// TwinCAT 3 PLC project PLC
// ProgramVersion: 3.1.4023.0
// libraries:
//   SPT Base Types, * (Beckhoff Automation LLC)
//   SPT XTS, * (Beckhoff Automation LLC)
//   Tc2_Standard, * (Beckhoff Automation GmbH)
//   Tc2_System, * (Beckhoff Automation GmbH)
//   Tc3_Module, * (Beckhoff Automation GmbH)
//   Tc3_PackML_V2, * (Beckhoff Automation GmbH)
//   Tc3_XTS_Utility, * (Beckhoff Automation GmbH)
// project tree:
//   / FB_Machine.TcPOU, PlcTask.TcTTO
//   POUs/ MAIN.TcPOU
// real-time tasks:
//   TASK XTS Task 1: cycle T#250us, priority 1, ADS port 350
//   TASK Job Task: cycle default, priority 32
//   TASK PlcTask: cycle T#10ms, priority 20, ADS port 351
// motion (NC):
//   TASK NC-Task 1: cycle T#2ms, priority 4, ADS port 501
//   TASK NC-Task 1 SVB: cycle T#10ms, priority 8, ADS port 511
//   AXIS Mover Axis 1 (id 1)
//     Dynamic: AccelerationMaximum=80000, DecelerationMaximum=80000, Acceleration=20000, Deceleration=20000, Jerk=200000
//     Velo: Maximum=4000
//     PositionAreaControl: Enable=false
//     TargetPosControl: Enable=false
//     OtherSettings: AllowMotionCmdToSlave=true, AllowMotionCmdToExtSetGenAxis=true
//     encoder EncType=28
//       EncPara: ModuloFactor=3000, ToleranceWndModuloStart=0.2, MaxCount=#xffffffff
//     drive DrvType=22
//       DrvPara: MaxCount=#xffffffff, DriveControlDWord=#x00000100
//         Analog: VeloReferenz=4200, TorqueSetpointScale=10
//         TimeComp: TaskDelayCycles=1
//     controller CtrType=1
//       CtrPara: PriorControlFactor=1
//         PosDiffControl: Range=10
//         Observer: BandWidth=20
//   AXIS Mover Axis 2 (id 2)
//     Dynamic: AccelerationMaximum=80000, DecelerationMaximum=80000, Acceleration=20000, Deceleration=20000, Jerk=200000
//     Velo: Maximum=4000
//     PositionAreaControl: Enable=false
//     TargetPosControl: Enable=false
//     OtherSettings: AllowMotionCmdToSlave=true, AllowMotionCmdToExtSetGenAxis=true
//     encoder EncType=28
//       EncPara: ModuloFactor=3000, ToleranceWndModuloStart=0.2, MaxCount=#xffffffff
//     drive DrvType=22
//       DrvPara: MaxCount=#xffffffff, DriveControlDWord=#x00000100
//         Analog: VeloReferenz=4200, TorqueSetpointScale=10
//         TimeComp: TaskDelayCycles=1
//     controller CtrType=1
//       CtrPara: PriorControlFactor=1
//         PosDiffControl: Range=10
//         Observer: BandWidth=20
//   AXIS Mover Axis 3 (id 3)
//     Dynamic: AccelerationMaximum=80000, DecelerationMaximum=80000, Acceleration=20000, Deceleration=20000, Jerk=200000
//     Velo: Maximum=4000
//     PositionAreaControl: Enable=false
//     TargetPosControl: Enable=false
//     OtherSettings: AllowMotionCmdToSlave=true, AllowMotionCmdToExtSetGenAxis=true
//     encoder EncType=28
//       EncPara: ModuloFactor=3000, ToleranceWndModuloStart=0.2, MaxCount=#xffffffff
//     drive DrvType=22
//       DrvPara: MaxCount=#xffffffff, DriveControlDWord=#x00000100
//         Analog: VeloReferenz=4200, TorqueSetpointScale=10
//         TimeComp: TaskDelayCycles=1
//     controller CtrType=1
//       CtrPara: PriorControlFactor=1
//         PosDiffControl: Range=10
//         Observer: BandWidth=20
//   AXIS Mover Axis 4 (id 4)
//     Dynamic: AccelerationMaximum=80000, DecelerationMaximum=80000, Acceleration=20000, Deceleration=20000, Jerk=200000
//     Velo: Maximum=4000
//     PositionAreaControl: Enable=false
//     TargetPosControl: Enable=false
//     OtherSettings: AllowMotionCmdToSlave=true, AllowMotionCmdToExtSetGenAxis=true
//     encoder EncType=28
//       EncPara: ModuloFactor=3000, ToleranceWndModuloStart=0.2, MaxCount=#xffffffff
//     drive DrvType=22
//       DrvPara: MaxCount=#xffffffff, DriveControlDWord=#x00000100
//         Analog: VeloReferenz=4200, TorqueSetpointScale=10
//         TimeComp: TaskDelayCycles=1
//     controller CtrType=1
//       CtrPara: PriorControlFactor=1
//         PosDiffControl: Range=10
//         Observer: BandWidth=20
//   AXIS Mover Axis 5 (id 5)
//     Dynamic: AccelerationMaximum=80000, DecelerationMaximum=80000, Acceleration=20000, Deceleration=20000, Jerk=200000
//     Velo: Maximum=4000
//     PositionAreaControl: Enable=false
//     TargetPosControl: Enable=false
//     OtherSettings: AllowMotionCmdToSlave=true, AllowMotionCmdToExtSetGenAxis=true
//     encoder EncType=28
//       EncPara: ModuloFactor=3000, ToleranceWndModuloStart=0.2, MaxCount=#xffffffff
//     drive DrvType=22
//       DrvPara: MaxCount=#xffffffff, DriveControlDWord=#x00000100
//         Analog: VeloReferenz=4200, TorqueSetpointScale=10
//         TimeComp: TaskDelayCycles=1
//     controller CtrType=1
//       CtrPara: PriorControlFactor=1
//         PosDiffControl: Range=10
//         Observer: BandWidth=20
//   AXIS Mover Axis 6 (id 6)
//     Dynamic: AccelerationMaximum=80000, DecelerationMaximum=80000, Acceleration=20000, Deceleration=20000, Jerk=200000
//     Velo: Maximum=4000
//     PositionAreaControl: Enable=false
//     TargetPosControl: Enable=false
//     OtherSettings: AllowMotionCmdToSlave=true, AllowMotionCmdToExtSetGenAxis=true
//     encoder EncType=28
//       EncPara: ModuloFactor=3000, ToleranceWndModuloStart=0.2, MaxCount=#xffffffff
//     drive DrvType=22
//       DrvPara: MaxCount=#xffffffff, DriveControlDWord=#x00000100
//         Analog: VeloReferenz=4200, TorqueSetpointScale=10
//         TimeComp: TaskDelayCycles=1
//     controller CtrType=1
//       CtrPara: PriorControlFactor=1
//         PosDiffControl: Range=10
//         Observer: BandWidth=20
//   AXIS Mover Axis 7 (id 7)
//     Dynamic: AccelerationMaximum=80000, DecelerationMaximum=80000, Acceleration=20000, Deceleration=20000, Jerk=200000
//     Velo: Maximum=4000
//     PositionAreaControl: Enable=false
//     TargetPosControl: Enable=false
//     OtherSettings: AllowMotionCmdToSlave=true, AllowMotionCmdToExtSetGenAxis=true
//     encoder EncType=28
//       EncPara: ModuloFactor=3000, ToleranceWndModuloStart=0.2, MaxCount=#xffffffff
//     drive DrvType=22
//       DrvPara: MaxCount=#xffffffff, DriveControlDWord=#x00000100
//         Analog: VeloReferenz=4200, TorqueSetpointScale=10
//         TimeComp: TaskDelayCycles=1
//     controller CtrType=1
//       CtrPara: PriorControlFactor=1
//         PosDiffControl: Range=10
//         Observer: BandWidth=20
//   AXIS Mover Axis 8 (id 8)
//     Dynamic: AccelerationMaximum=80000, DecelerationMaximum=80000, Acceleration=20000, Deceleration=20000, Jerk=200000
//     Velo: Maximum=4000
//     PositionAreaControl: Enable=false
//     TargetPosControl: Enable=false
//     OtherSettings: AllowMotionCmdToSlave=true, AllowMotionCmdToExtSetGenAxis=true
//     encoder EncType=28
//       EncPara: ModuloFactor=3000, ToleranceWndModuloStart=0.2, MaxCount=#xffffffff
//     drive DrvType=22
//       DrvPara: MaxCount=#xffffffff, DriveControlDWord=#x00000100
//         Analog: VeloReferenz=4200, TorqueSetpointScale=10
//         TimeComp: TaskDelayCycles=1
//     controller CtrType=1
//       CtrPara: PriorControlFactor=1
//         PosDiffControl: Range=10
//         Observer: BandWidth=20
//   AXIS Mover Axis 9 (id 9)
//     Dynamic: AccelerationMaximum=80000, DecelerationMaximum=80000, Acceleration=20000, Deceleration=20000, Jerk=200000
//     Velo: Maximum=4000
//     PositionAreaControl: Enable=false
//     TargetPosControl: Enable=false
//     OtherSettings: AllowMotionCmdToSlave=true, AllowMotionCmdToExtSetGenAxis=true
//     encoder EncType=28
//       EncPara: ModuloFactor=3000, ToleranceWndModuloStart=0.2, MaxCount=#xffffffff
//     drive DrvType=22
//       DrvPara: MaxCount=#xffffffff, DriveControlDWord=#x00000100
//         Analog: VeloReferenz=4200, TorqueSetpointScale=10
//         TimeComp: TaskDelayCycles=1
//     controller CtrType=1
//       CtrPara: PriorControlFactor=1
//         PosDiffControl: Range=10
//         Observer: BandWidth=20
//   AXIS Mover Axis 10 (id 10)
//     Dynamic: AccelerationMaximum=80000, DecelerationMaximum=80000, Acceleration=20000, Deceleration=20000, Jerk=200000
//     Velo: Maximum=4000
//     PositionAreaControl: Enable=false
//     TargetPosControl: Enable=false
//     OtherSettings: AllowMotionCmdToSlave=true, AllowMotionCmdToExtSetGenAxis=true
//     encoder EncType=28
//       EncPara: ModuloFactor=3000, ToleranceWndModuloStart=0.2, MaxCount=#xffffffff
//     drive DrvType=22
//       DrvPara: MaxCount=#xffffffff, DriveControlDWord=#x00000100
//         Analog: VeloReferenz=4200, TorqueSetpointScale=10
//         TimeComp: TaskDelayCycles=1
//     controller CtrType=1
//       CtrPara: PriorControlFactor=1
//         PosDiffControl: Range=10
//         Observer: BandWidth=20
// I/O:
//   DEVICE Device 1 (disabled), AmsNetId 192.168.111.1.2.1
//     Term 1 (AT2001-0250) [AT2001-0250 Motor module with feed 250 mm, 48V]
//       Term 2 (AT2001-5250) [AT2001-5250 Sensor line with feed]
//     Term 3 (AT2000-0250) [AT2000-0250 Motor module 250 mm, 48V]
//       Term 4 (AT2000-5250) [AT2000-5250 Sensor line]
//     Term 5 (AT2000-0250) [AT2000-0250 Motor module 250 mm, 48V]
//       Term 6 (AT2000-5250) [AT2000-5250 Sensor line]
//     Term 7 (AT2000-0250) [AT2000-0250 Motor module 250 mm, 48V]
//       Term 8 (AT2000-5250) [AT2000-5250 Sensor line]
//     Term 9 (AT2050-0500) [AT2050-0500 Motor module, 90° clothoid, EtherCAT In, 48V]
//       Term 10 (AT2050-5500) [AT2050-5500 Sensor line 90° clothoid, EtherCAT In]
//     Term 11 (AT2050-0501) [AT2050-0501 Motor module, 90° clothoid, EtherCAT Out, 48V]
//       Term 12 (AT2050-5501) [AT2050-5501 Sensor line 90° clothoid, EtherCAT Out]
//   DEVICE Device 2 (disabled), AmsNetId 192.168.111.1.3.1
//     Term 13 (AT2001-0250) [AT2001-0250 Motor module with feed 250 mm, 48V]
//       Term 14 (AT2001-5250) [AT2001-5250 Sensor line with feed]
//     Term 15 (AT2000-0250) [AT2000-0250 Motor module 250 mm, 48V]
//       Term 16 (AT2000-5250) [AT2000-5250 Sensor line]
//     Term 17 (AT2000-0250) [AT2000-0250 Motor module 250 mm, 48V]
//       Term 18 (AT2000-5250) [AT2000-5250 Sensor line]
//     Term 19 (AT2000-0250) [AT2000-0250 Motor module 250 mm, 48V]
//       Term 20 (AT2000-5250) [AT2000-5250 Sensor line]
//     Term 21 (AT2050-0500) [AT2050-0500 Motor module, 90° clothoid, EtherCAT In, 48V]
//       Term 22 (AT2050-5500) [AT2050-5500 Sensor line 90° clothoid, EtherCAT In]
//     Term 23 (AT2050-0501) [AT2050-0501 Motor module, 90° clothoid, EtherCAT Out, 48V]
//       Term 24 (AT2050-5501) [AT2050-5501 Sensor line 90° clothoid, EtherCAT Out]
// variable links:
//   Device 1 <-> TcCOM Objects/XtsProcessingUnit 1/Part 1/Module 1
//     Term 1 (AT2001-0250)/CC Inputs/Current actual value Ch.1 <-> Data Pointer/CurrentActualValues[0]
//     Term 1 (AT2001-0250)/CC Inputs/Current actual value Ch.10 <-> Data Pointer/CurrentActualValues[9]
//     Term 1 (AT2001-0250)/CC Inputs/Current actual value Ch.11 <-> Data Pointer/CurrentActualValues[10]
//     Term 1 (AT2001-0250)/CC Inputs/Current actual value Ch.12 <-> Data Pointer/CurrentActualValues[11]
//     Term 1 (AT2001-0250)/CC Inputs/Current actual value Ch.13 <-> Data Pointer/CurrentActualValues[12]
//     Term 1 (AT2001-0250)/CC Inputs/Current actual value Ch.14 <-> Data Pointer/CurrentActualValues[13]
//     Term 1 (AT2001-0250)/CC Inputs/Current actual value Ch.15 <-> Data Pointer/CurrentActualValues[14]
//     Term 1 (AT2001-0250)/CC Inputs/Current actual value Ch.2 <-> Data Pointer/CurrentActualValues[1]
//     Term 1 (AT2001-0250)/CC Inputs/Current actual value Ch.3 <-> Data Pointer/CurrentActualValues[2]
//     Term 1 (AT2001-0250)/CC Inputs/Current actual value Ch.4 <-> Data Pointer/CurrentActualValues[3]
//     Term 1 (AT2001-0250)/CC Inputs/Current actual value Ch.5 <-> Data Pointer/CurrentActualValues[4]
//     Term 1 (AT2001-0250)/CC Inputs/Current actual value Ch.6 <-> Data Pointer/CurrentActualValues[5]
//     Term 1 (AT2001-0250)/CC Inputs/Current actual value Ch.7 <-> Data Pointer/CurrentActualValues[6]
//     Term 1 (AT2001-0250)/CC Inputs/Current actual value Ch.8 <-> Data Pointer/CurrentActualValues[7]
//     Term 1 (AT2001-0250)/CC Inputs/Current actual value Ch.9 <-> Data Pointer/CurrentActualValues[8]
//     Term 1 (AT2001-0250)/CC Inputs/Status <-> Data Pointer/Status
//     Term 1 (AT2001-0250)/CC Outputs/Control <-> Data Pointer/Control
//     Term 1 (AT2001-0250)/CC Outputs/Current setpoint value Ch.1 <-> Data Pointer/CurrentSetpointValues[0]
//     Term 1 (AT2001-0250)/CC Outputs/Current setpoint value Ch.10 <-> Data Pointer/CurrentSetpointValues[9]
//     Term 1 (AT2001-0250)/CC Outputs/Current setpoint value Ch.11 <-> Data Pointer/CurrentSetpointValues[10]
//     Term 1 (AT2001-0250)/CC Outputs/Current setpoint value Ch.12 <-> Data Pointer/CurrentSetpointValues[11]
//     Term 1 (AT2001-0250)/CC Outputs/Current setpoint value Ch.13 <-> Data Pointer/CurrentSetpointValues[12]
//     Term 1 (AT2001-0250)/CC Outputs/Current setpoint value Ch.14 <-> Data Pointer/CurrentSetpointValues[13]
//     Term 1 (AT2001-0250)/CC Outputs/Current setpoint value Ch.15 <-> Data Pointer/CurrentSetpointValues[14]
//     Term 1 (AT2001-0250)/CC Outputs/Current setpoint value Ch.2 <-> Data Pointer/CurrentSetpointValues[1]
//     Term 1 (AT2001-0250)/CC Outputs/Current setpoint value Ch.3 <-> Data Pointer/CurrentSetpointValues[2]
//     Term 1 (AT2001-0250)/CC Outputs/Current setpoint value Ch.4 <-> Data Pointer/CurrentSetpointValues[3]
//     Term 1 (AT2001-0250)/CC Outputs/Current setpoint value Ch.5 <-> Data Pointer/CurrentSetpointValues[4]
//     Term 1 (AT2001-0250)/CC Outputs/Current setpoint value Ch.6 <-> Data Pointer/CurrentSetpointValues[5]
//     Term 1 (AT2001-0250)/CC Outputs/Current setpoint value Ch.7 <-> Data Pointer/CurrentSetpointValues[6]
//     Term 1 (AT2001-0250)/CC Outputs/Current setpoint value Ch.8 <-> Data Pointer/CurrentSetpointValues[7]
//     Term 1 (AT2001-0250)/CC Outputs/Current setpoint value Ch.9 <-> Data Pointer/CurrentSetpointValues[8]
//     Term 1 (AT2001-0250)/Term 2 (AT2001-5250)/FB Inputs/Value Channel 01 <-> Data Pointer/RawPositionValues[0]
//     Term 1 (AT2001-0250)/Term 2 (AT2001-5250)/FB Inputs/Value Channel 02 <-> Data Pointer/RawPositionValues[1]
//     Term 1 (AT2001-0250)/Term 2 (AT2001-5250)/FB Inputs/Value Channel 03 <-> Data Pointer/RawPositionValues[2]
//     Term 1 (AT2001-0250)/Term 2 (AT2001-5250)/FB Inputs/Value Channel 04 <-> Data Pointer/RawPositionValues[3]
//     Term 1 (AT2001-0250)/Term 2 (AT2001-5250)/FB Inputs/Value Channel 05 <-> Data Pointer/RawPositionValues[4]
//     Term 1 (AT2001-0250)/Term 2 (AT2001-5250)/FB Inputs/Value Channel 06 <-> Data Pointer/RawPositionValues[5]
//     Term 1 (AT2001-0250)/Term 2 (AT2001-5250)/FB Inputs/Value Channel 07 <-> Data Pointer/RawPositionValues[6]
//     Term 1 (AT2001-0250)/Term 2 (AT2001-5250)/FB Inputs/Value Channel 08 <-> Data Pointer/RawPositionValues[7]
//     Term 1 (AT2001-0250)/Term 2 (AT2001-5250)/FB Inputs/Value Channel 09 <-> Data Pointer/RawPositionValues[8]
//     Term 1 (AT2001-0250)/Term 2 (AT2001-5250)/FB Inputs/Value Channel 10 <-> Data Pointer/RawPositionValues[9]
//     Term 1 (AT2001-0250)/Term 2 (AT2001-5250)/FB Inputs/Value Channel 11 <-> Data Pointer/RawPositionValues[10]
//     Term 1 (AT2001-0250)/Term 2 (AT2001-5250)/FB Inputs/Value Channel 12 <-> Data Pointer/RawPositionValues[11]
//     Term 1 (AT2001-0250)/Term 2 (AT2001-5250)/FB Inputs/Value Channel 13 <-> Data Pointer/RawPositionValues[12]
//     Term 1 (AT2001-0250)/Term 2 (AT2001-5250)/FB Inputs/Value Channel 14 <-> Data Pointer/RawPositionValues[13]
//     Term 1 (AT2001-0250)/Term 2 (AT2001-5250)/FB Inputs/Value Channel 15 <-> Data Pointer/RawPositionValues[14]
//     Term 1 (AT2001-0250)/Term 2 (AT2001-5250)/FB Inputs/Value Channel 16 <-> Data Pointer/RawPositionValues[15]
//     Term 1 (AT2001-0250)/Term 2 (AT2001-5250)/FB Inputs/Value Channel 17 <-> Data Pointer/RawPositionValues[16]
//     Term 1 (AT2001-0250)/Term 2 (AT2001-5250)/FB Inputs/Value Channel 18 <-> Data Pointer/RawPositionValues[17]
//     Term 1 (AT2001-0250)/Term 2 (AT2001-5250)/FB Inputs/Value Channel 19 <-> Data Pointer/RawPositionValues[18]
//     Term 1 (AT2001-0250)/Term 2 (AT2001-5250)/FB Inputs/Value Channel 20 <-> Data Pointer/RawPositionValues[19]
//     Term 1 (AT2001-0250)/Term 2 (AT2001-5250)/FB Inputs/Value Channel 21 <-> Data Pointer/RawPositionValues[20]
//     Term 1 (AT2001-0250)/Term 2 (AT2001-5250)/FB Inputs/Value Channel 22 <-> Data Pointer/RawPositionValues[21]
//     Term 1 (AT2001-0250)/Term 2 (AT2001-5250)/FB Inputs/Value Channel 23 <-> Data Pointer/RawPositionValues[22]
//     Term 1 (AT2001-0250)/Term 2 (AT2001-5250)/FB Inputs/Value Channel 24 <-> Data Pointer/RawPositionValues[23]
//     Term 1 (AT2001-0250)/Term 2 (AT2001-5250)/FB Inputs/Value Channel 25 <-> Data Pointer/RawPositionValues[24]
//     Term 1 (AT2001-0250)/Term 2 (AT2001-5250)/FB Inputs/Value Channel 26 <-> Data Pointer/RawPositionValues[25]
//     Term 1 (AT2001-0250)/Term 2 (AT2001-5250)/FB Inputs/Value Channel 27 <-> Data Pointer/RawPositionValues[26]
//     Term 1 (AT2001-0250)/Term 2 (AT2001-5250)/FB Inputs/Value Channel 28 <-> Data Pointer/RawPositionValues[27]
//     Term 1 (AT2001-0250)/Term 2 (AT2001-5250)/FB Inputs/Value Channel 29 <-> Data Pointer/RawPositionValues[28]
//     Term 1 (AT2001-0250)/Term 2 (AT2001-5250)/FB Inputs/Value Channel 30 <-> Data Pointer/RawPositionValues[29]
//     Term 1 (AT2001-0250)/Term 2 (AT2001-5250)/FB Inputs/Value Channel 31 <-> Data Pointer/RawPositionValues[30]
//     Term 1 (AT2001-0250)/Term 2 (AT2001-5250)/FB Inputs/Value Channel 32 <-> Data Pointer/RawPositionValues[31]
//   Device 1 <-> TcCOM Objects/XtsProcessingUnit 1/Part 1/Module 2
//     Term 3 (AT2000-0250)/CC Inputs/Current actual value Ch.1 <-> Data Pointer/CurrentActualValues[0]
//     Term 3 (AT2000-0250)/CC Inputs/Current actual value Ch.10 <-> Data Pointer/CurrentActualValues[9]
//     Term 3 (AT2000-0250)/CC Inputs/Current actual value Ch.11 <-> Data Pointer/CurrentActualValues[10]
//     Term 3 (AT2000-0250)/CC Inputs/Current actual value Ch.12 <-> Data Pointer/CurrentActualValues[11]
//     Term 3 (AT2000-0250)/CC Inputs/Current actual value Ch.13 <-> Data Pointer/CurrentActualValues[12]
//     Term 3 (AT2000-0250)/CC Inputs/Current actual value Ch.14 <-> Data Pointer/CurrentActualValues[13]
//     Term 3 (AT2000-0250)/CC Inputs/Current actual value Ch.15 <-> Data Pointer/CurrentActualValues[14]
//     Term 3 (AT2000-0250)/CC Inputs/Current actual value Ch.2 <-> Data Pointer/CurrentActualValues[1]
//     Term 3 (AT2000-0250)/CC Inputs/Current actual value Ch.3 <-> Data Pointer/CurrentActualValues[2]
//     Term 3 (AT2000-0250)/CC Inputs/Current actual value Ch.4 <-> Data Pointer/CurrentActualValues[3]
//     Term 3 (AT2000-0250)/CC Inputs/Current actual value Ch.5 <-> Data Pointer/CurrentActualValues[4]
//     Term 3 (AT2000-0250)/CC Inputs/Current actual value Ch.6 <-> Data Pointer/CurrentActualValues[5]
//     Term 3 (AT2000-0250)/CC Inputs/Current actual value Ch.7 <-> Data Pointer/CurrentActualValues[6]
//     Term 3 (AT2000-0250)/CC Inputs/Current actual value Ch.8 <-> Data Pointer/CurrentActualValues[7]
//     Term 3 (AT2000-0250)/CC Inputs/Current actual value Ch.9 <-> Data Pointer/CurrentActualValues[8]
//     Term 3 (AT2000-0250)/CC Inputs/Status <-> Data Pointer/Status
//     Term 3 (AT2000-0250)/CC Outputs/Control <-> Data Pointer/Control
//     Term 3 (AT2000-0250)/CC Outputs/Current setpoint value Ch.1 <-> Data Pointer/CurrentSetpointValues[0]
//     Term 3 (AT2000-0250)/CC Outputs/Current setpoint value Ch.10 <-> Data Pointer/CurrentSetpointValues[9]
//     Term 3 (AT2000-0250)/CC Outputs/Current setpoint value Ch.11 <-> Data Pointer/CurrentSetpointValues[10]
//     Term 3 (AT2000-0250)/CC Outputs/Current setpoint value Ch.12 <-> Data Pointer/CurrentSetpointValues[11]
//     Term 3 (AT2000-0250)/CC Outputs/Current setpoint value Ch.13 <-> Data Pointer/CurrentSetpointValues[12]
//     Term 3 (AT2000-0250)/CC Outputs/Current setpoint value Ch.14 <-> Data Pointer/CurrentSetpointValues[13]
//     Term 3 (AT2000-0250)/CC Outputs/Current setpoint value Ch.15 <-> Data Pointer/CurrentSetpointValues[14]
//     Term 3 (AT2000-0250)/CC Outputs/Current setpoint value Ch.2 <-> Data Pointer/CurrentSetpointValues[1]
//     Term 3 (AT2000-0250)/CC Outputs/Current setpoint value Ch.3 <-> Data Pointer/CurrentSetpointValues[2]
//     Term 3 (AT2000-0250)/CC Outputs/Current setpoint value Ch.4 <-> Data Pointer/CurrentSetpointValues[3]
//     Term 3 (AT2000-0250)/CC Outputs/Current setpoint value Ch.5 <-> Data Pointer/CurrentSetpointValues[4]
//     Term 3 (AT2000-0250)/CC Outputs/Current setpoint value Ch.6 <-> Data Pointer/CurrentSetpointValues[5]
//     Term 3 (AT2000-0250)/CC Outputs/Current setpoint value Ch.7 <-> Data Pointer/CurrentSetpointValues[6]
//     Term 3 (AT2000-0250)/CC Outputs/Current setpoint value Ch.8 <-> Data Pointer/CurrentSetpointValues[7]
//     Term 3 (AT2000-0250)/CC Outputs/Current setpoint value Ch.9 <-> Data Pointer/CurrentSetpointValues[8]
//     Term 3 (AT2000-0250)/Term 4 (AT2000-5250)/FB Inputs/Value Channel 01 <-> Data Pointer/RawPositionValues[0]
//     Term 3 (AT2000-0250)/Term 4 (AT2000-5250)/FB Inputs/Value Channel 02 <-> Data Pointer/RawPositionValues[1]
//     Term 3 (AT2000-0250)/Term 4 (AT2000-5250)/FB Inputs/Value Channel 03 <-> Data Pointer/RawPositionValues[2]
//     Term 3 (AT2000-0250)/Term 4 (AT2000-5250)/FB Inputs/Value Channel 04 <-> Data Pointer/RawPositionValues[3]
//     Term 3 (AT2000-0250)/Term 4 (AT2000-5250)/FB Inputs/Value Channel 05 <-> Data Pointer/RawPositionValues[4]
//     Term 3 (AT2000-0250)/Term 4 (AT2000-5250)/FB Inputs/Value Channel 06 <-> Data Pointer/RawPositionValues[5]
//     Term 3 (AT2000-0250)/Term 4 (AT2000-5250)/FB Inputs/Value Channel 07 <-> Data Pointer/RawPositionValues[6]
//     Term 3 (AT2000-0250)/Term 4 (AT2000-5250)/FB Inputs/Value Channel 08 <-> Data Pointer/RawPositionValues[7]
//     Term 3 (AT2000-0250)/Term 4 (AT2000-5250)/FB Inputs/Value Channel 09 <-> Data Pointer/RawPositionValues[8]
//     Term 3 (AT2000-0250)/Term 4 (AT2000-5250)/FB Inputs/Value Channel 10 <-> Data Pointer/RawPositionValues[9]
//     Term 3 (AT2000-0250)/Term 4 (AT2000-5250)/FB Inputs/Value Channel 11 <-> Data Pointer/RawPositionValues[10]
//     Term 3 (AT2000-0250)/Term 4 (AT2000-5250)/FB Inputs/Value Channel 12 <-> Data Pointer/RawPositionValues[11]
//     Term 3 (AT2000-0250)/Term 4 (AT2000-5250)/FB Inputs/Value Channel 13 <-> Data Pointer/RawPositionValues[12]
//     Term 3 (AT2000-0250)/Term 4 (AT2000-5250)/FB Inputs/Value Channel 14 <-> Data Pointer/RawPositionValues[13]
//     Term 3 (AT2000-0250)/Term 4 (AT2000-5250)/FB Inputs/Value Channel 15 <-> Data Pointer/RawPositionValues[14]
//     Term 3 (AT2000-0250)/Term 4 (AT2000-5250)/FB Inputs/Value Channel 16 <-> Data Pointer/RawPositionValues[15]
//     Term 3 (AT2000-0250)/Term 4 (AT2000-5250)/FB Inputs/Value Channel 17 <-> Data Pointer/RawPositionValues[16]
//     Term 3 (AT2000-0250)/Term 4 (AT2000-5250)/FB Inputs/Value Channel 18 <-> Data Pointer/RawPositionValues[17]
//     Term 3 (AT2000-0250)/Term 4 (AT2000-5250)/FB Inputs/Value Channel 19 <-> Data Pointer/RawPositionValues[18]
//     Term 3 (AT2000-0250)/Term 4 (AT2000-5250)/FB Inputs/Value Channel 20 <-> Data Pointer/RawPositionValues[19]
//     Term 3 (AT2000-0250)/Term 4 (AT2000-5250)/FB Inputs/Value Channel 21 <-> Data Pointer/RawPositionValues[20]
//     Term 3 (AT2000-0250)/Term 4 (AT2000-5250)/FB Inputs/Value Channel 22 <-> Data Pointer/RawPositionValues[21]
//     Term 3 (AT2000-0250)/Term 4 (AT2000-5250)/FB Inputs/Value Channel 23 <-> Data Pointer/RawPositionValues[22]
//     Term 3 (AT2000-0250)/Term 4 (AT2000-5250)/FB Inputs/Value Channel 24 <-> Data Pointer/RawPositionValues[23]
//     Term 3 (AT2000-0250)/Term 4 (AT2000-5250)/FB Inputs/Value Channel 25 <-> Data Pointer/RawPositionValues[24]
//     Term 3 (AT2000-0250)/Term 4 (AT2000-5250)/FB Inputs/Value Channel 26 <-> Data Pointer/RawPositionValues[25]
//     Term 3 (AT2000-0250)/Term 4 (AT2000-5250)/FB Inputs/Value Channel 27 <-> Data Pointer/RawPositionValues[26]
//     Term 3 (AT2000-0250)/Term 4 (AT2000-5250)/FB Inputs/Value Channel 28 <-> Data Pointer/RawPositionValues[27]
//     Term 3 (AT2000-0250)/Term 4 (AT2000-5250)/FB Inputs/Value Channel 29 <-> Data Pointer/RawPositionValues[28]
//     Term 3 (AT2000-0250)/Term 4 (AT2000-5250)/FB Inputs/Value Channel 30 <-> Data Pointer/RawPositionValues[29]
//     Term 3 (AT2000-0250)/Term 4 (AT2000-5250)/FB Inputs/Value Channel 31 <-> Data Pointer/RawPositionValues[30]
//     Term 3 (AT2000-0250)/Term 4 (AT2000-5250)/FB Inputs/Value Channel 32 <-> Data Pointer/RawPositionValues[31]
//   Device 1 <-> TcCOM Objects/XtsProcessingUnit 1/Part 1/Module 3
//     Term 5 (AT2000-0250)/CC Inputs/Current actual value Ch.1 <-> Data Pointer/CurrentActualValues[0]
//     Term 5 (AT2000-0250)/CC Inputs/Current actual value Ch.10 <-> Data Pointer/CurrentActualValues[9]
//     Term 5 (AT2000-0250)/CC Inputs/Current actual value Ch.11 <-> Data Pointer/CurrentActualValues[10]
//     Term 5 (AT2000-0250)/CC Inputs/Current actual value Ch.12 <-> Data Pointer/CurrentActualValues[11]
//     Term 5 (AT2000-0250)/CC Inputs/Current actual value Ch.13 <-> Data Pointer/CurrentActualValues[12]
//     Term 5 (AT2000-0250)/CC Inputs/Current actual value Ch.14 <-> Data Pointer/CurrentActualValues[13]
//     Term 5 (AT2000-0250)/CC Inputs/Current actual value Ch.15 <-> Data Pointer/CurrentActualValues[14]
//     Term 5 (AT2000-0250)/CC Inputs/Current actual value Ch.2 <-> Data Pointer/CurrentActualValues[1]
//     Term 5 (AT2000-0250)/CC Inputs/Current actual value Ch.3 <-> Data Pointer/CurrentActualValues[2]
//     Term 5 (AT2000-0250)/CC Inputs/Current actual value Ch.4 <-> Data Pointer/CurrentActualValues[3]
//     Term 5 (AT2000-0250)/CC Inputs/Current actual value Ch.5 <-> Data Pointer/CurrentActualValues[4]
//     Term 5 (AT2000-0250)/CC Inputs/Current actual value Ch.6 <-> Data Pointer/CurrentActualValues[5]
//     Term 5 (AT2000-0250)/CC Inputs/Current actual value Ch.7 <-> Data Pointer/CurrentActualValues[6]
//     Term 5 (AT2000-0250)/CC Inputs/Current actual value Ch.8 <-> Data Pointer/CurrentActualValues[7]
//     Term 5 (AT2000-0250)/CC Inputs/Current actual value Ch.9 <-> Data Pointer/CurrentActualValues[8]
//     Term 5 (AT2000-0250)/CC Inputs/Status <-> Data Pointer/Status
//     Term 5 (AT2000-0250)/CC Outputs/Control <-> Data Pointer/Control
//     Term 5 (AT2000-0250)/CC Outputs/Current setpoint value Ch.1 <-> Data Pointer/CurrentSetpointValues[0]
//     Term 5 (AT2000-0250)/CC Outputs/Current setpoint value Ch.10 <-> Data Pointer/CurrentSetpointValues[9]
//     Term 5 (AT2000-0250)/CC Outputs/Current setpoint value Ch.11 <-> Data Pointer/CurrentSetpointValues[10]
//     Term 5 (AT2000-0250)/CC Outputs/Current setpoint value Ch.12 <-> Data Pointer/CurrentSetpointValues[11]
//     Term 5 (AT2000-0250)/CC Outputs/Current setpoint value Ch.13 <-> Data Pointer/CurrentSetpointValues[12]
//     Term 5 (AT2000-0250)/CC Outputs/Current setpoint value Ch.14 <-> Data Pointer/CurrentSetpointValues[13]
//     Term 5 (AT2000-0250)/CC Outputs/Current setpoint value Ch.15 <-> Data Pointer/CurrentSetpointValues[14]
//     Term 5 (AT2000-0250)/CC Outputs/Current setpoint value Ch.2 <-> Data Pointer/CurrentSetpointValues[1]
//     Term 5 (AT2000-0250)/CC Outputs/Current setpoint value Ch.3 <-> Data Pointer/CurrentSetpointValues[2]
//     Term 5 (AT2000-0250)/CC Outputs/Current setpoint value Ch.4 <-> Data Pointer/CurrentSetpointValues[3]
//     Term 5 (AT2000-0250)/CC Outputs/Current setpoint value Ch.5 <-> Data Pointer/CurrentSetpointValues[4]
//     Term 5 (AT2000-0250)/CC Outputs/Current setpoint value Ch.6 <-> Data Pointer/CurrentSetpointValues[5]
//     Term 5 (AT2000-0250)/CC Outputs/Current setpoint value Ch.7 <-> Data Pointer/CurrentSetpointValues[6]
//     Term 5 (AT2000-0250)/CC Outputs/Current setpoint value Ch.8 <-> Data Pointer/CurrentSetpointValues[7]
//     Term 5 (AT2000-0250)/CC Outputs/Current setpoint value Ch.9 <-> Data Pointer/CurrentSetpointValues[8]
//     Term 5 (AT2000-0250)/Term 6 (AT2000-5250)/FB Inputs/Value Channel 01 <-> Data Pointer/RawPositionValues[0]
//     Term 5 (AT2000-0250)/Term 6 (AT2000-5250)/FB Inputs/Value Channel 02 <-> Data Pointer/RawPositionValues[1]
//     Term 5 (AT2000-0250)/Term 6 (AT2000-5250)/FB Inputs/Value Channel 03 <-> Data Pointer/RawPositionValues[2]
//     Term 5 (AT2000-0250)/Term 6 (AT2000-5250)/FB Inputs/Value Channel 04 <-> Data Pointer/RawPositionValues[3]
//     Term 5 (AT2000-0250)/Term 6 (AT2000-5250)/FB Inputs/Value Channel 05 <-> Data Pointer/RawPositionValues[4]
//     Term 5 (AT2000-0250)/Term 6 (AT2000-5250)/FB Inputs/Value Channel 06 <-> Data Pointer/RawPositionValues[5]
//     Term 5 (AT2000-0250)/Term 6 (AT2000-5250)/FB Inputs/Value Channel 07 <-> Data Pointer/RawPositionValues[6]
//     Term 5 (AT2000-0250)/Term 6 (AT2000-5250)/FB Inputs/Value Channel 08 <-> Data Pointer/RawPositionValues[7]
//     Term 5 (AT2000-0250)/Term 6 (AT2000-5250)/FB Inputs/Value Channel 09 <-> Data Pointer/RawPositionValues[8]
//     Term 5 (AT2000-0250)/Term 6 (AT2000-5250)/FB Inputs/Value Channel 10 <-> Data Pointer/RawPositionValues[9]
//     Term 5 (AT2000-0250)/Term 6 (AT2000-5250)/FB Inputs/Value Channel 11 <-> Data Pointer/RawPositionValues[10]
//     Term 5 (AT2000-0250)/Term 6 (AT2000-5250)/FB Inputs/Value Channel 12 <-> Data Pointer/RawPositionValues[11]
//     Term 5 (AT2000-0250)/Term 6 (AT2000-5250)/FB Inputs/Value Channel 13 <-> Data Pointer/RawPositionValues[12]
//     Term 5 (AT2000-0250)/Term 6 (AT2000-5250)/FB Inputs/Value Channel 14 <-> Data Pointer/RawPositionValues[13]
//     Term 5 (AT2000-0250)/Term 6 (AT2000-5250)/FB Inputs/Value Channel 15 <-> Data Pointer/RawPositionValues[14]
//     Term 5 (AT2000-0250)/Term 6 (AT2000-5250)/FB Inputs/Value Channel 16 <-> Data Pointer/RawPositionValues[15]
//     Term 5 (AT2000-0250)/Term 6 (AT2000-5250)/FB Inputs/Value Channel 17 <-> Data Pointer/RawPositionValues[16]
//     Term 5 (AT2000-0250)/Term 6 (AT2000-5250)/FB Inputs/Value Channel 18 <-> Data Pointer/RawPositionValues[17]
//     Term 5 (AT2000-0250)/Term 6 (AT2000-5250)/FB Inputs/Value Channel 19 <-> Data Pointer/RawPositionValues[18]
//     Term 5 (AT2000-0250)/Term 6 (AT2000-5250)/FB Inputs/Value Channel 20 <-> Data Pointer/RawPositionValues[19]
//     Term 5 (AT2000-0250)/Term 6 (AT2000-5250)/FB Inputs/Value Channel 21 <-> Data Pointer/RawPositionValues[20]
//     Term 5 (AT2000-0250)/Term 6 (AT2000-5250)/FB Inputs/Value Channel 22 <-> Data Pointer/RawPositionValues[21]
//     Term 5 (AT2000-0250)/Term 6 (AT2000-5250)/FB Inputs/Value Channel 23 <-> Data Pointer/RawPositionValues[22]
//     Term 5 (AT2000-0250)/Term 6 (AT2000-5250)/FB Inputs/Value Channel 24 <-> Data Pointer/RawPositionValues[23]
//     Term 5 (AT2000-0250)/Term 6 (AT2000-5250)/FB Inputs/Value Channel 25 <-> Data Pointer/RawPositionValues[24]
//     Term 5 (AT2000-0250)/Term 6 (AT2000-5250)/FB Inputs/Value Channel 26 <-> Data Pointer/RawPositionValues[25]
//     Term 5 (AT2000-0250)/Term 6 (AT2000-5250)/FB Inputs/Value Channel 27 <-> Data Pointer/RawPositionValues[26]
//     Term 5 (AT2000-0250)/Term 6 (AT2000-5250)/FB Inputs/Value Channel 28 <-> Data Pointer/RawPositionValues[27]
//     Term 5 (AT2000-0250)/Term 6 (AT2000-5250)/FB Inputs/Value Channel 29 <-> Data Pointer/RawPositionValues[28]
//     Term 5 (AT2000-0250)/Term 6 (AT2000-5250)/FB Inputs/Value Channel 30 <-> Data Pointer/RawPositionValues[29]
//     Term 5 (AT2000-0250)/Term 6 (AT2000-5250)/FB Inputs/Value Channel 31 <-> Data Pointer/RawPositionValues[30]
//     Term 5 (AT2000-0250)/Term 6 (AT2000-5250)/FB Inputs/Value Channel 32 <-> Data Pointer/RawPositionValues[31]
//   Device 1 <-> TcCOM Objects/XtsProcessingUnit 1/Part 1/Module 4
//     Term 7 (AT2000-0250)/CC Inputs/Current actual value Ch.1 <-> Data Pointer/CurrentActualValues[0]
//     Term 7 (AT2000-0250)/CC Inputs/Current actual value Ch.10 <-> Data Pointer/CurrentActualValues[9]
//     Term 7 (AT2000-0250)/CC Inputs/Current actual value Ch.11 <-> Data Pointer/CurrentActualValues[10]
//     Term 7 (AT2000-0250)/CC Inputs/Current actual value Ch.12 <-> Data Pointer/CurrentActualValues[11]
//     Term 7 (AT2000-0250)/CC Inputs/Current actual value Ch.13 <-> Data Pointer/CurrentActualValues[12]
//     Term 7 (AT2000-0250)/CC Inputs/Current actual value Ch.14 <-> Data Pointer/CurrentActualValues[13]
//     Term 7 (AT2000-0250)/CC Inputs/Current actual value Ch.15 <-> Data Pointer/CurrentActualValues[14]
//     Term 7 (AT2000-0250)/CC Inputs/Current actual value Ch.2 <-> Data Pointer/CurrentActualValues[1]
//     Term 7 (AT2000-0250)/CC Inputs/Current actual value Ch.3 <-> Data Pointer/CurrentActualValues[2]
//     Term 7 (AT2000-0250)/CC Inputs/Current actual value Ch.4 <-> Data Pointer/CurrentActualValues[3]
//     Term 7 (AT2000-0250)/CC Inputs/Current actual value Ch.5 <-> Data Pointer/CurrentActualValues[4]
//     Term 7 (AT2000-0250)/CC Inputs/Current actual value Ch.6 <-> Data Pointer/CurrentActualValues[5]
//     Term 7 (AT2000-0250)/CC Inputs/Current actual value Ch.7 <-> Data Pointer/CurrentActualValues[6]
//     Term 7 (AT2000-0250)/CC Inputs/Current actual value Ch.8 <-> Data Pointer/CurrentActualValues[7]
//     Term 7 (AT2000-0250)/CC Inputs/Current actual value Ch.9 <-> Data Pointer/CurrentActualValues[8]
//     Term 7 (AT2000-0250)/CC Inputs/Status <-> Data Pointer/Status
//     Term 7 (AT2000-0250)/CC Outputs/Control <-> Data Pointer/Control
//     Term 7 (AT2000-0250)/CC Outputs/Current setpoint value Ch.1 <-> Data Pointer/CurrentSetpointValues[0]
//     Term 7 (AT2000-0250)/CC Outputs/Current setpoint value Ch.10 <-> Data Pointer/CurrentSetpointValues[9]
//     Term 7 (AT2000-0250)/CC Outputs/Current setpoint value Ch.11 <-> Data Pointer/CurrentSetpointValues[10]
//     Term 7 (AT2000-0250)/CC Outputs/Current setpoint value Ch.12 <-> Data Pointer/CurrentSetpointValues[11]
//     Term 7 (AT2000-0250)/CC Outputs/Current setpoint value Ch.13 <-> Data Pointer/CurrentSetpointValues[12]
//     Term 7 (AT2000-0250)/CC Outputs/Current setpoint value Ch.14 <-> Data Pointer/CurrentSetpointValues[13]
//     Term 7 (AT2000-0250)/CC Outputs/Current setpoint value Ch.15 <-> Data Pointer/CurrentSetpointValues[14]
//     Term 7 (AT2000-0250)/CC Outputs/Current setpoint value Ch.2 <-> Data Pointer/CurrentSetpointValues[1]
//     Term 7 (AT2000-0250)/CC Outputs/Current setpoint value Ch.3 <-> Data Pointer/CurrentSetpointValues[2]
//     Term 7 (AT2000-0250)/CC Outputs/Current setpoint value Ch.4 <-> Data Pointer/CurrentSetpointValues[3]
//     Term 7 (AT2000-0250)/CC Outputs/Current setpoint value Ch.5 <-> Data Pointer/CurrentSetpointValues[4]
//     Term 7 (AT2000-0250)/CC Outputs/Current setpoint value Ch.6 <-> Data Pointer/CurrentSetpointValues[5]
//     Term 7 (AT2000-0250)/CC Outputs/Current setpoint value Ch.7 <-> Data Pointer/CurrentSetpointValues[6]
//     Term 7 (AT2000-0250)/CC Outputs/Current setpoint value Ch.8 <-> Data Pointer/CurrentSetpointValues[7]
//     Term 7 (AT2000-0250)/CC Outputs/Current setpoint value Ch.9 <-> Data Pointer/CurrentSetpointValues[8]
//     Term 7 (AT2000-0250)/Term 8 (AT2000-5250)/FB Inputs/Value Channel 01 <-> Data Pointer/RawPositionValues[0]
//     Term 7 (AT2000-0250)/Term 8 (AT2000-5250)/FB Inputs/Value Channel 02 <-> Data Pointer/RawPositionValues[1]
//     Term 7 (AT2000-0250)/Term 8 (AT2000-5250)/FB Inputs/Value Channel 03 <-> Data Pointer/RawPositionValues[2]
//     Term 7 (AT2000-0250)/Term 8 (AT2000-5250)/FB Inputs/Value Channel 04 <-> Data Pointer/RawPositionValues[3]
//     Term 7 (AT2000-0250)/Term 8 (AT2000-5250)/FB Inputs/Value Channel 05 <-> Data Pointer/RawPositionValues[4]
//     Term 7 (AT2000-0250)/Term 8 (AT2000-5250)/FB Inputs/Value Channel 06 <-> Data Pointer/RawPositionValues[5]
//     Term 7 (AT2000-0250)/Term 8 (AT2000-5250)/FB Inputs/Value Channel 07 <-> Data Pointer/RawPositionValues[6]
//     Term 7 (AT2000-0250)/Term 8 (AT2000-5250)/FB Inputs/Value Channel 08 <-> Data Pointer/RawPositionValues[7]
//     Term 7 (AT2000-0250)/Term 8 (AT2000-5250)/FB Inputs/Value Channel 09 <-> Data Pointer/RawPositionValues[8]
//     Term 7 (AT2000-0250)/Term 8 (AT2000-5250)/FB Inputs/Value Channel 10 <-> Data Pointer/RawPositionValues[9]
//     Term 7 (AT2000-0250)/Term 8 (AT2000-5250)/FB Inputs/Value Channel 11 <-> Data Pointer/RawPositionValues[10]
//     Term 7 (AT2000-0250)/Term 8 (AT2000-5250)/FB Inputs/Value Channel 12 <-> Data Pointer/RawPositionValues[11]
//     Term 7 (AT2000-0250)/Term 8 (AT2000-5250)/FB Inputs/Value Channel 13 <-> Data Pointer/RawPositionValues[12]
//     Term 7 (AT2000-0250)/Term 8 (AT2000-5250)/FB Inputs/Value Channel 14 <-> Data Pointer/RawPositionValues[13]
//     Term 7 (AT2000-0250)/Term 8 (AT2000-5250)/FB Inputs/Value Channel 15 <-> Data Pointer/RawPositionValues[14]
//     Term 7 (AT2000-0250)/Term 8 (AT2000-5250)/FB Inputs/Value Channel 16 <-> Data Pointer/RawPositionValues[15]
//     Term 7 (AT2000-0250)/Term 8 (AT2000-5250)/FB Inputs/Value Channel 17 <-> Data Pointer/RawPositionValues[16]
//     Term 7 (AT2000-0250)/Term 8 (AT2000-5250)/FB Inputs/Value Channel 18 <-> Data Pointer/RawPositionValues[17]
//     Term 7 (AT2000-0250)/Term 8 (AT2000-5250)/FB Inputs/Value Channel 19 <-> Data Pointer/RawPositionValues[18]
//     Term 7 (AT2000-0250)/Term 8 (AT2000-5250)/FB Inputs/Value Channel 20 <-> Data Pointer/RawPositionValues[19]
//     Term 7 (AT2000-0250)/Term 8 (AT2000-5250)/FB Inputs/Value Channel 21 <-> Data Pointer/RawPositionValues[20]
//     Term 7 (AT2000-0250)/Term 8 (AT2000-5250)/FB Inputs/Value Channel 22 <-> Data Pointer/RawPositionValues[21]
//     Term 7 (AT2000-0250)/Term 8 (AT2000-5250)/FB Inputs/Value Channel 23 <-> Data Pointer/RawPositionValues[22]
//     Term 7 (AT2000-0250)/Term 8 (AT2000-5250)/FB Inputs/Value Channel 24 <-> Data Pointer/RawPositionValues[23]
//     Term 7 (AT2000-0250)/Term 8 (AT2000-5250)/FB Inputs/Value Channel 25 <-> Data Pointer/RawPositionValues[24]
//     Term 7 (AT2000-0250)/Term 8 (AT2000-5250)/FB Inputs/Value Channel 26 <-> Data Pointer/RawPositionValues[25]
//     Term 7 (AT2000-0250)/Term 8 (AT2000-5250)/FB Inputs/Value Channel 27 <-> Data Pointer/RawPositionValues[26]
//     Term 7 (AT2000-0250)/Term 8 (AT2000-5250)/FB Inputs/Value Channel 28 <-> Data Pointer/RawPositionValues[27]
//     Term 7 (AT2000-0250)/Term 8 (AT2000-5250)/FB Inputs/Value Channel 29 <-> Data Pointer/RawPositionValues[28]
//     Term 7 (AT2000-0250)/Term 8 (AT2000-5250)/FB Inputs/Value Channel 30 <-> Data Pointer/RawPositionValues[29]
//     Term 7 (AT2000-0250)/Term 8 (AT2000-5250)/FB Inputs/Value Channel 31 <-> Data Pointer/RawPositionValues[30]
//     Term 7 (AT2000-0250)/Term 8 (AT2000-5250)/FB Inputs/Value Channel 32 <-> Data Pointer/RawPositionValues[31]
//   Device 1 <-> TcCOM Objects/XtsProcessingUnit 1/Part 1/Module 5
//     Term 9 (AT2050-0500)/CC Inputs/Current actual value Ch.1 <-> Data Pointer/CurrentActualValues[0]
//     Term 9 (AT2050-0500)/CC Inputs/Current actual value Ch.10 <-> Data Pointer/CurrentActualValues[9]
//     Term 9 (AT2050-0500)/CC Inputs/Current actual value Ch.11 <-> Data Pointer/CurrentActualValues[10]
//     Term 9 (AT2050-0500)/CC Inputs/Current actual value Ch.12 <-> Data Pointer/CurrentActualValues[11]
//     Term 9 (AT2050-0500)/CC Inputs/Current actual value Ch.13 <-> Data Pointer/CurrentActualValues[12]
//     Term 9 (AT2050-0500)/CC Inputs/Current actual value Ch.14 <-> Data Pointer/CurrentActualValues[13]
//     Term 9 (AT2050-0500)/CC Inputs/Current actual value Ch.15 <-> Data Pointer/CurrentActualValues[14]
//     Term 9 (AT2050-0500)/CC Inputs/Current actual value Ch.2 <-> Data Pointer/CurrentActualValues[1]
//     Term 9 (AT2050-0500)/CC Inputs/Current actual value Ch.3 <-> Data Pointer/CurrentActualValues[2]
//     Term 9 (AT2050-0500)/CC Inputs/Current actual value Ch.4 <-> Data Pointer/CurrentActualValues[3]
//     Term 9 (AT2050-0500)/CC Inputs/Current actual value Ch.5 <-> Data Pointer/CurrentActualValues[4]
//     Term 9 (AT2050-0500)/CC Inputs/Current actual value Ch.6 <-> Data Pointer/CurrentActualValues[5]
//     Term 9 (AT2050-0500)/CC Inputs/Current actual value Ch.7 <-> Data Pointer/CurrentActualValues[6]
//     Term 9 (AT2050-0500)/CC Inputs/Current actual value Ch.8 <-> Data Pointer/CurrentActualValues[7]
//     Term 9 (AT2050-0500)/CC Inputs/Current actual value Ch.9 <-> Data Pointer/CurrentActualValues[8]
//     Term 9 (AT2050-0500)/CC Inputs/Status <-> Data Pointer/Status
//     Term 9 (AT2050-0500)/CC Outputs/Control <-> Data Pointer/Control
//     Term 9 (AT2050-0500)/CC Outputs/Current setpoint value Ch.1 <-> Data Pointer/CurrentSetpointValues[0]
//     Term 9 (AT2050-0500)/CC Outputs/Current setpoint value Ch.10 <-> Data Pointer/CurrentSetpointValues[9]
//     Term 9 (AT2050-0500)/CC Outputs/Current setpoint value Ch.11 <-> Data Pointer/CurrentSetpointValues[10]
//     Term 9 (AT2050-0500)/CC Outputs/Current setpoint value Ch.12 <-> Data Pointer/CurrentSetpointValues[11]
//     Term 9 (AT2050-0500)/CC Outputs/Current setpoint value Ch.13 <-> Data Pointer/CurrentSetpointValues[12]
//     Term 9 (AT2050-0500)/CC Outputs/Current setpoint value Ch.14 <-> Data Pointer/CurrentSetpointValues[13]
//     Term 9 (AT2050-0500)/CC Outputs/Current setpoint value Ch.15 <-> Data Pointer/CurrentSetpointValues[14]
//     Term 9 (AT2050-0500)/CC Outputs/Current setpoint value Ch.2 <-> Data Pointer/CurrentSetpointValues[1]
//     Term 9 (AT2050-0500)/CC Outputs/Current setpoint value Ch.3 <-> Data Pointer/CurrentSetpointValues[2]
//     Term 9 (AT2050-0500)/CC Outputs/Current setpoint value Ch.4 <-> Data Pointer/CurrentSetpointValues[3]
//     Term 9 (AT2050-0500)/CC Outputs/Current setpoint value Ch.5 <-> Data Pointer/CurrentSetpointValues[4]
//     Term 9 (AT2050-0500)/CC Outputs/Current setpoint value Ch.6 <-> Data Pointer/CurrentSetpointValues[5]
//     Term 9 (AT2050-0500)/CC Outputs/Current setpoint value Ch.7 <-> Data Pointer/CurrentSetpointValues[6]
//     Term 9 (AT2050-0500)/CC Outputs/Current setpoint value Ch.8 <-> Data Pointer/CurrentSetpointValues[7]
//     Term 9 (AT2050-0500)/CC Outputs/Current setpoint value Ch.9 <-> Data Pointer/CurrentSetpointValues[8]
//     Term 9 (AT2050-0500)/Term 10 (AT2050-5500)/FB Inputs/Value Channel 01 <-> Data Pointer/RawPositionValues[0]
//     Term 9 (AT2050-0500)/Term 10 (AT2050-5500)/FB Inputs/Value Channel 02 <-> Data Pointer/RawPositionValues[1]
//     Term 9 (AT2050-0500)/Term 10 (AT2050-5500)/FB Inputs/Value Channel 03 <-> Data Pointer/RawPositionValues[2]
//     Term 9 (AT2050-0500)/Term 10 (AT2050-5500)/FB Inputs/Value Channel 04 <-> Data Pointer/RawPositionValues[3]
//     Term 9 (AT2050-0500)/Term 10 (AT2050-5500)/FB Inputs/Value Channel 05 <-> Data Pointer/RawPositionValues[4]
//     Term 9 (AT2050-0500)/Term 10 (AT2050-5500)/FB Inputs/Value Channel 06 <-> Data Pointer/RawPositionValues[5]
//     Term 9 (AT2050-0500)/Term 10 (AT2050-5500)/FB Inputs/Value Channel 07 <-> Data Pointer/RawPositionValues[6]
//     Term 9 (AT2050-0500)/Term 10 (AT2050-5500)/FB Inputs/Value Channel 08 <-> Data Pointer/RawPositionValues[7]
//     Term 9 (AT2050-0500)/Term 10 (AT2050-5500)/FB Inputs/Value Channel 09 <-> Data Pointer/RawPositionValues[8]
//     Term 9 (AT2050-0500)/Term 10 (AT2050-5500)/FB Inputs/Value Channel 10 <-> Data Pointer/RawPositionValues[9]
//     Term 9 (AT2050-0500)/Term 10 (AT2050-5500)/FB Inputs/Value Channel 11 <-> Data Pointer/RawPositionValues[10]
//     Term 9 (AT2050-0500)/Term 10 (AT2050-5500)/FB Inputs/Value Channel 12 <-> Data Pointer/RawPositionValues[11]
//     Term 9 (AT2050-0500)/Term 10 (AT2050-5500)/FB Inputs/Value Channel 13 <-> Data Pointer/RawPositionValues[12]
//     Term 9 (AT2050-0500)/Term 10 (AT2050-5500)/FB Inputs/Value Channel 14 <-> Data Pointer/RawPositionValues[13]
//     Term 9 (AT2050-0500)/Term 10 (AT2050-5500)/FB Inputs/Value Channel 15 <-> Data Pointer/RawPositionValues[14]
//     Term 9 (AT2050-0500)/Term 10 (AT2050-5500)/FB Inputs/Value Channel 16 <-> Data Pointer/RawPositionValues[15]
//     Term 9 (AT2050-0500)/Term 10 (AT2050-5500)/FB Inputs/Value Channel 17 <-> Data Pointer/RawPositionValues[16]
//     Term 9 (AT2050-0500)/Term 10 (AT2050-5500)/FB Inputs/Value Channel 18 <-> Data Pointer/RawPositionValues[17]
//     Term 9 (AT2050-0500)/Term 10 (AT2050-5500)/FB Inputs/Value Channel 19 <-> Data Pointer/RawPositionValues[18]
//     Term 9 (AT2050-0500)/Term 10 (AT2050-5500)/FB Inputs/Value Channel 20 <-> Data Pointer/RawPositionValues[19]
//     Term 9 (AT2050-0500)/Term 10 (AT2050-5500)/FB Inputs/Value Channel 21 <-> Data Pointer/RawPositionValues[20]
//     Term 9 (AT2050-0500)/Term 10 (AT2050-5500)/FB Inputs/Value Channel 22 <-> Data Pointer/RawPositionValues[21]
//     Term 9 (AT2050-0500)/Term 10 (AT2050-5500)/FB Inputs/Value Channel 23 <-> Data Pointer/RawPositionValues[22]
//     Term 9 (AT2050-0500)/Term 10 (AT2050-5500)/FB Inputs/Value Channel 24 <-> Data Pointer/RawPositionValues[23]
//     Term 9 (AT2050-0500)/Term 10 (AT2050-5500)/FB Inputs/Value Channel 25 <-> Data Pointer/RawPositionValues[24]
//     Term 9 (AT2050-0500)/Term 10 (AT2050-5500)/FB Inputs/Value Channel 26 <-> Data Pointer/RawPositionValues[25]
//     Term 9 (AT2050-0500)/Term 10 (AT2050-5500)/FB Inputs/Value Channel 27 <-> Data Pointer/RawPositionValues[26]
//     Term 9 (AT2050-0500)/Term 10 (AT2050-5500)/FB Inputs/Value Channel 28 <-> Data Pointer/RawPositionValues[27]
//     Term 9 (AT2050-0500)/Term 10 (AT2050-5500)/FB Inputs/Value Channel 29 <-> Data Pointer/RawPositionValues[28]
//     Term 9 (AT2050-0500)/Term 10 (AT2050-5500)/FB Inputs/Value Channel 30 <-> Data Pointer/RawPositionValues[29]
//     Term 9 (AT2050-0500)/Term 10 (AT2050-5500)/FB Inputs/Value Channel 31 <-> Data Pointer/RawPositionValues[30]
//     Term 9 (AT2050-0500)/Term 10 (AT2050-5500)/FB Inputs/Value Channel 32 <-> Data Pointer/RawPositionValues[31]
//   Device 1 <-> TcCOM Objects/XtsProcessingUnit 1/Part 1/Module 6
//     Term 11 (AT2050-0501)/CC Inputs/Current actual value Ch.1 <-> Data Pointer/CurrentActualValues[0]
//     Term 11 (AT2050-0501)/CC Inputs/Current actual value Ch.10 <-> Data Pointer/CurrentActualValues[9]
//     Term 11 (AT2050-0501)/CC Inputs/Current actual value Ch.11 <-> Data Pointer/CurrentActualValues[10]
//     Term 11 (AT2050-0501)/CC Inputs/Current actual value Ch.12 <-> Data Pointer/CurrentActualValues[11]
//     Term 11 (AT2050-0501)/CC Inputs/Current actual value Ch.13 <-> Data Pointer/CurrentActualValues[12]
//     Term 11 (AT2050-0501)/CC Inputs/Current actual value Ch.14 <-> Data Pointer/CurrentActualValues[13]
//     Term 11 (AT2050-0501)/CC Inputs/Current actual value Ch.15 <-> Data Pointer/CurrentActualValues[14]
//     Term 11 (AT2050-0501)/CC Inputs/Current actual value Ch.2 <-> Data Pointer/CurrentActualValues[1]
//     Term 11 (AT2050-0501)/CC Inputs/Current actual value Ch.3 <-> Data Pointer/CurrentActualValues[2]
//     Term 11 (AT2050-0501)/CC Inputs/Current actual value Ch.4 <-> Data Pointer/CurrentActualValues[3]
//     Term 11 (AT2050-0501)/CC Inputs/Current actual value Ch.5 <-> Data Pointer/CurrentActualValues[4]
//     Term 11 (AT2050-0501)/CC Inputs/Current actual value Ch.6 <-> Data Pointer/CurrentActualValues[5]
//     Term 11 (AT2050-0501)/CC Inputs/Current actual value Ch.7 <-> Data Pointer/CurrentActualValues[6]
//     Term 11 (AT2050-0501)/CC Inputs/Current actual value Ch.8 <-> Data Pointer/CurrentActualValues[7]
//     Term 11 (AT2050-0501)/CC Inputs/Current actual value Ch.9 <-> Data Pointer/CurrentActualValues[8]
//     Term 11 (AT2050-0501)/CC Inputs/Status <-> Data Pointer/Status
//     Term 11 (AT2050-0501)/CC Outputs/Control <-> Data Pointer/Control
//     Term 11 (AT2050-0501)/CC Outputs/Current setpoint value Ch.1 <-> Data Pointer/CurrentSetpointValues[0]
//     Term 11 (AT2050-0501)/CC Outputs/Current setpoint value Ch.10 <-> Data Pointer/CurrentSetpointValues[9]
//     Term 11 (AT2050-0501)/CC Outputs/Current setpoint value Ch.11 <-> Data Pointer/CurrentSetpointValues[10]
//     Term 11 (AT2050-0501)/CC Outputs/Current setpoint value Ch.12 <-> Data Pointer/CurrentSetpointValues[11]
//     Term 11 (AT2050-0501)/CC Outputs/Current setpoint value Ch.13 <-> Data Pointer/CurrentSetpointValues[12]
//     Term 11 (AT2050-0501)/CC Outputs/Current setpoint value Ch.14 <-> Data Pointer/CurrentSetpointValues[13]
//     Term 11 (AT2050-0501)/CC Outputs/Current setpoint value Ch.15 <-> Data Pointer/CurrentSetpointValues[14]
//     Term 11 (AT2050-0501)/CC Outputs/Current setpoint value Ch.2 <-> Data Pointer/CurrentSetpointValues[1]
//     Term 11 (AT2050-0501)/CC Outputs/Current setpoint value Ch.3 <-> Data Pointer/CurrentSetpointValues[2]
//     Term 11 (AT2050-0501)/CC Outputs/Current setpoint value Ch.4 <-> Data Pointer/CurrentSetpointValues[3]
//     Term 11 (AT2050-0501)/CC Outputs/Current setpoint value Ch.5 <-> Data Pointer/CurrentSetpointValues[4]
//     Term 11 (AT2050-0501)/CC Outputs/Current setpoint value Ch.6 <-> Data Pointer/CurrentSetpointValues[5]
//     Term 11 (AT2050-0501)/CC Outputs/Current setpoint value Ch.7 <-> Data Pointer/CurrentSetpointValues[6]
//     Term 11 (AT2050-0501)/CC Outputs/Current setpoint value Ch.8 <-> Data Pointer/CurrentSetpointValues[7]
//     Term 11 (AT2050-0501)/CC Outputs/Current setpoint value Ch.9 <-> Data Pointer/CurrentSetpointValues[8]
//     Term 11 (AT2050-0501)/Term 12 (AT2050-5501)/FB Inputs/Value Channel 01 <-> Data Pointer/RawPositionValues[0]
//     Term 11 (AT2050-0501)/Term 12 (AT2050-5501)/FB Inputs/Value Channel 02 <-> Data Pointer/RawPositionValues[1]
//     Term 11 (AT2050-0501)/Term 12 (AT2050-5501)/FB Inputs/Value Channel 03 <-> Data Pointer/RawPositionValues[2]
//     Term 11 (AT2050-0501)/Term 12 (AT2050-5501)/FB Inputs/Value Channel 04 <-> Data Pointer/RawPositionValues[3]
//     Term 11 (AT2050-0501)/Term 12 (AT2050-5501)/FB Inputs/Value Channel 05 <-> Data Pointer/RawPositionValues[4]
//     Term 11 (AT2050-0501)/Term 12 (AT2050-5501)/FB Inputs/Value Channel 06 <-> Data Pointer/RawPositionValues[5]
//     Term 11 (AT2050-0501)/Term 12 (AT2050-5501)/FB Inputs/Value Channel 07 <-> Data Pointer/RawPositionValues[6]
//     Term 11 (AT2050-0501)/Term 12 (AT2050-5501)/FB Inputs/Value Channel 08 <-> Data Pointer/RawPositionValues[7]
//     Term 11 (AT2050-0501)/Term 12 (AT2050-5501)/FB Inputs/Value Channel 09 <-> Data Pointer/RawPositionValues[8]
//     Term 11 (AT2050-0501)/Term 12 (AT2050-5501)/FB Inputs/Value Channel 10 <-> Data Pointer/RawPositionValues[9]
//     Term 11 (AT2050-0501)/Term 12 (AT2050-5501)/FB Inputs/Value Channel 11 <-> Data Pointer/RawPositionValues[10]
//     Term 11 (AT2050-0501)/Term 12 (AT2050-5501)/FB Inputs/Value Channel 12 <-> Data Pointer/RawPositionValues[11]
//     Term 11 (AT2050-0501)/Term 12 (AT2050-5501)/FB Inputs/Value Channel 13 <-> Data Pointer/RawPositionValues[12]
//     Term 11 (AT2050-0501)/Term 12 (AT2050-5501)/FB Inputs/Value Channel 14 <-> Data Pointer/RawPositionValues[13]
//     Term 11 (AT2050-0501)/Term 12 (AT2050-5501)/FB Inputs/Value Channel 15 <-> Data Pointer/RawPositionValues[14]
//     Term 11 (AT2050-0501)/Term 12 (AT2050-5501)/FB Inputs/Value Channel 16 <-> Data Pointer/RawPositionValues[15]
//     Term 11 (AT2050-0501)/Term 12 (AT2050-5501)/FB Inputs/Value Channel 17 <-> Data Pointer/RawPositionValues[16]
//     Term 11 (AT2050-0501)/Term 12 (AT2050-5501)/FB Inputs/Value Channel 18 <-> Data Pointer/RawPositionValues[17]
//     Term 11 (AT2050-0501)/Term 12 (AT2050-5501)/FB Inputs/Value Channel 19 <-> Data Pointer/RawPositionValues[18]
//     Term 11 (AT2050-0501)/Term 12 (AT2050-5501)/FB Inputs/Value Channel 20 <-> Data Pointer/RawPositionValues[19]
//     Term 11 (AT2050-0501)/Term 12 (AT2050-5501)/FB Inputs/Value Channel 21 <-> Data Pointer/RawPositionValues[20]
//     Term 11 (AT2050-0501)/Term 12 (AT2050-5501)/FB Inputs/Value Channel 22 <-> Data Pointer/RawPositionValues[21]
//     Term 11 (AT2050-0501)/Term 12 (AT2050-5501)/FB Inputs/Value Channel 23 <-> Data Pointer/RawPositionValues[22]
//     Term 11 (AT2050-0501)/Term 12 (AT2050-5501)/FB Inputs/Value Channel 24 <-> Data Pointer/RawPositionValues[23]
//     Term 11 (AT2050-0501)/Term 12 (AT2050-5501)/FB Inputs/Value Channel 25 <-> Data Pointer/RawPositionValues[24]
//     Term 11 (AT2050-0501)/Term 12 (AT2050-5501)/FB Inputs/Value Channel 26 <-> Data Pointer/RawPositionValues[25]
//     Term 11 (AT2050-0501)/Term 12 (AT2050-5501)/FB Inputs/Value Channel 27 <-> Data Pointer/RawPositionValues[26]
//     Term 11 (AT2050-0501)/Term 12 (AT2050-5501)/FB Inputs/Value Channel 28 <-> Data Pointer/RawPositionValues[27]
//     Term 11 (AT2050-0501)/Term 12 (AT2050-5501)/FB Inputs/Value Channel 29 <-> Data Pointer/RawPositionValues[28]
//     Term 11 (AT2050-0501)/Term 12 (AT2050-5501)/FB Inputs/Value Channel 30 <-> Data Pointer/RawPositionValues[29]
//     Term 11 (AT2050-0501)/Term 12 (AT2050-5501)/FB Inputs/Value Channel 31 <-> Data Pointer/RawPositionValues[30]
//     Term 11 (AT2050-0501)/Term 12 (AT2050-5501)/FB Inputs/Value Channel 32 <-> Data Pointer/RawPositionValues[31]
//   Device 2 <-> TcCOM Objects/XtsProcessingUnit 1/Part 1/Module 10
//     Term 19 (AT2000-0250)/CC Inputs/Current actual value Ch.1 <-> Data Pointer/CurrentActualValues[0]
//     Term 19 (AT2000-0250)/CC Inputs/Current actual value Ch.10 <-> Data Pointer/CurrentActualValues[9]
//     Term 19 (AT2000-0250)/CC Inputs/Current actual value Ch.11 <-> Data Pointer/CurrentActualValues[10]
//     Term 19 (AT2000-0250)/CC Inputs/Current actual value Ch.12 <-> Data Pointer/CurrentActualValues[11]
//     Term 19 (AT2000-0250)/CC Inputs/Current actual value Ch.13 <-> Data Pointer/CurrentActualValues[12]
//     Term 19 (AT2000-0250)/CC Inputs/Current actual value Ch.14 <-> Data Pointer/CurrentActualValues[13]
//     Term 19 (AT2000-0250)/CC Inputs/Current actual value Ch.15 <-> Data Pointer/CurrentActualValues[14]
//     Term 19 (AT2000-0250)/CC Inputs/Current actual value Ch.2 <-> Data Pointer/CurrentActualValues[1]
//     Term 19 (AT2000-0250)/CC Inputs/Current actual value Ch.3 <-> Data Pointer/CurrentActualValues[2]
//     Term 19 (AT2000-0250)/CC Inputs/Current actual value Ch.4 <-> Data Pointer/CurrentActualValues[3]
//     Term 19 (AT2000-0250)/CC Inputs/Current actual value Ch.5 <-> Data Pointer/CurrentActualValues[4]
//     Term 19 (AT2000-0250)/CC Inputs/Current actual value Ch.6 <-> Data Pointer/CurrentActualValues[5]
//     Term 19 (AT2000-0250)/CC Inputs/Current actual value Ch.7 <-> Data Pointer/CurrentActualValues[6]
//     Term 19 (AT2000-0250)/CC Inputs/Current actual value Ch.8 <-> Data Pointer/CurrentActualValues[7]
//     Term 19 (AT2000-0250)/CC Inputs/Current actual value Ch.9 <-> Data Pointer/CurrentActualValues[8]
//     Term 19 (AT2000-0250)/CC Inputs/Status <-> Data Pointer/Status
//     Term 19 (AT2000-0250)/CC Outputs/Control <-> Data Pointer/Control
//     Term 19 (AT2000-0250)/CC Outputs/Current setpoint value Ch.1 <-> Data Pointer/CurrentSetpointValues[0]
//     Term 19 (AT2000-0250)/CC Outputs/Current setpoint value Ch.10 <-> Data Pointer/CurrentSetpointValues[9]
//     Term 19 (AT2000-0250)/CC Outputs/Current setpoint value Ch.11 <-> Data Pointer/CurrentSetpointValues[10]
//     Term 19 (AT2000-0250)/CC Outputs/Current setpoint value Ch.12 <-> Data Pointer/CurrentSetpointValues[11]
//     Term 19 (AT2000-0250)/CC Outputs/Current setpoint value Ch.13 <-> Data Pointer/CurrentSetpointValues[12]
//     Term 19 (AT2000-0250)/CC Outputs/Current setpoint value Ch.14 <-> Data Pointer/CurrentSetpointValues[13]
//     Term 19 (AT2000-0250)/CC Outputs/Current setpoint value Ch.15 <-> Data Pointer/CurrentSetpointValues[14]
//     Term 19 (AT2000-0250)/CC Outputs/Current setpoint value Ch.2 <-> Data Pointer/CurrentSetpointValues[1]
//     Term 19 (AT2000-0250)/CC Outputs/Current setpoint value Ch.3 <-> Data Pointer/CurrentSetpointValues[2]
//     Term 19 (AT2000-0250)/CC Outputs/Current setpoint value Ch.4 <-> Data Pointer/CurrentSetpointValues[3]
//     Term 19 (AT2000-0250)/CC Outputs/Current setpoint value Ch.5 <-> Data Pointer/CurrentSetpointValues[4]
//     Term 19 (AT2000-0250)/CC Outputs/Current setpoint value Ch.6 <-> Data Pointer/CurrentSetpointValues[5]
//     Term 19 (AT2000-0250)/CC Outputs/Current setpoint value Ch.7 <-> Data Pointer/CurrentSetpointValues[6]
//     Term 19 (AT2000-0250)/CC Outputs/Current setpoint value Ch.8 <-> Data Pointer/CurrentSetpointValues[7]
//     Term 19 (AT2000-0250)/CC Outputs/Current setpoint value Ch.9 <-> Data Pointer/CurrentSetpointValues[8]
//     Term 19 (AT2000-0250)/Term 20 (AT2000-5250)/FB Inputs/Value Channel 01 <-> Data Pointer/RawPositionValues[0]
//     Term 19 (AT2000-0250)/Term 20 (AT2000-5250)/FB Inputs/Value Channel 02 <-> Data Pointer/RawPositionValues[1]
//     Term 19 (AT2000-0250)/Term 20 (AT2000-5250)/FB Inputs/Value Channel 03 <-> Data Pointer/RawPositionValues[2]
//     Term 19 (AT2000-0250)/Term 20 (AT2000-5250)/FB Inputs/Value Channel 04 <-> Data Pointer/RawPositionValues[3]
//     Term 19 (AT2000-0250)/Term 20 (AT2000-5250)/FB Inputs/Value Channel 05 <-> Data Pointer/RawPositionValues[4]
//     Term 19 (AT2000-0250)/Term 20 (AT2000-5250)/FB Inputs/Value Channel 06 <-> Data Pointer/RawPositionValues[5]
//     Term 19 (AT2000-0250)/Term 20 (AT2000-5250)/FB Inputs/Value Channel 07 <-> Data Pointer/RawPositionValues[6]
//     Term 19 (AT2000-0250)/Term 20 (AT2000-5250)/FB Inputs/Value Channel 08 <-> Data Pointer/RawPositionValues[7]
//     Term 19 (AT2000-0250)/Term 20 (AT2000-5250)/FB Inputs/Value Channel 09 <-> Data Pointer/RawPositionValues[8]
//     Term 19 (AT2000-0250)/Term 20 (AT2000-5250)/FB Inputs/Value Channel 10 <-> Data Pointer/RawPositionValues[9]
//     Term 19 (AT2000-0250)/Term 20 (AT2000-5250)/FB Inputs/Value Channel 11 <-> Data Pointer/RawPositionValues[10]
//     Term 19 (AT2000-0250)/Term 20 (AT2000-5250)/FB Inputs/Value Channel 12 <-> Data Pointer/RawPositionValues[11]
//     Term 19 (AT2000-0250)/Term 20 (AT2000-5250)/FB Inputs/Value Channel 13 <-> Data Pointer/RawPositionValues[12]
//     Term 19 (AT2000-0250)/Term 20 (AT2000-5250)/FB Inputs/Value Channel 14 <-> Data Pointer/RawPositionValues[13]
//     Term 19 (AT2000-0250)/Term 20 (AT2000-5250)/FB Inputs/Value Channel 15 <-> Data Pointer/RawPositionValues[14]
//     Term 19 (AT2000-0250)/Term 20 (AT2000-5250)/FB Inputs/Value Channel 16 <-> Data Pointer/RawPositionValues[15]
//     Term 19 (AT2000-0250)/Term 20 (AT2000-5250)/FB Inputs/Value Channel 17 <-> Data Pointer/RawPositionValues[16]
//     Term 19 (AT2000-0250)/Term 20 (AT2000-5250)/FB Inputs/Value Channel 18 <-> Data Pointer/RawPositionValues[17]
//     Term 19 (AT2000-0250)/Term 20 (AT2000-5250)/FB Inputs/Value Channel 19 <-> Data Pointer/RawPositionValues[18]
//     Term 19 (AT2000-0250)/Term 20 (AT2000-5250)/FB Inputs/Value Channel 20 <-> Data Pointer/RawPositionValues[19]
//     Term 19 (AT2000-0250)/Term 20 (AT2000-5250)/FB Inputs/Value Channel 21 <-> Data Pointer/RawPositionValues[20]
//     Term 19 (AT2000-0250)/Term 20 (AT2000-5250)/FB Inputs/Value Channel 22 <-> Data Pointer/RawPositionValues[21]
//     Term 19 (AT2000-0250)/Term 20 (AT2000-5250)/FB Inputs/Value Channel 23 <-> Data Pointer/RawPositionValues[22]
//     Term 19 (AT2000-0250)/Term 20 (AT2000-5250)/FB Inputs/Value Channel 24 <-> Data Pointer/RawPositionValues[23]
//     Term 19 (AT2000-0250)/Term 20 (AT2000-5250)/FB Inputs/Value Channel 25 <-> Data Pointer/RawPositionValues[24]
//     Term 19 (AT2000-0250)/Term 20 (AT2000-5250)/FB Inputs/Value Channel 26 <-> Data Pointer/RawPositionValues[25]
//     Term 19 (AT2000-0250)/Term 20 (AT2000-5250)/FB Inputs/Value Channel 27 <-> Data Pointer/RawPositionValues[26]
//     Term 19 (AT2000-0250)/Term 20 (AT2000-5250)/FB Inputs/Value Channel 28 <-> Data Pointer/RawPositionValues[27]
//     Term 19 (AT2000-0250)/Term 20 (AT2000-5250)/FB Inputs/Value Channel 29 <-> Data Pointer/RawPositionValues[28]
//     Term 19 (AT2000-0250)/Term 20 (AT2000-5250)/FB Inputs/Value Channel 30 <-> Data Pointer/RawPositionValues[29]
//     Term 19 (AT2000-0250)/Term 20 (AT2000-5250)/FB Inputs/Value Channel 31 <-> Data Pointer/RawPositionValues[30]
//     Term 19 (AT2000-0250)/Term 20 (AT2000-5250)/FB Inputs/Value Channel 32 <-> Data Pointer/RawPositionValues[31]
//   Device 2 <-> TcCOM Objects/XtsProcessingUnit 1/Part 1/Module 11
//     Term 21 (AT2050-0500)/CC Inputs/Current actual value Ch.1 <-> Data Pointer/CurrentActualValues[0]
//     Term 21 (AT2050-0500)/CC Inputs/Current actual value Ch.10 <-> Data Pointer/CurrentActualValues[9]
//     Term 21 (AT2050-0500)/CC Inputs/Current actual value Ch.11 <-> Data Pointer/CurrentActualValues[10]
//     Term 21 (AT2050-0500)/CC Inputs/Current actual value Ch.12 <-> Data Pointer/CurrentActualValues[11]
//     Term 21 (AT2050-0500)/CC Inputs/Current actual value Ch.13 <-> Data Pointer/CurrentActualValues[12]
//     Term 21 (AT2050-0500)/CC Inputs/Current actual value Ch.14 <-> Data Pointer/CurrentActualValues[13]
//     Term 21 (AT2050-0500)/CC Inputs/Current actual value Ch.15 <-> Data Pointer/CurrentActualValues[14]
//     Term 21 (AT2050-0500)/CC Inputs/Current actual value Ch.2 <-> Data Pointer/CurrentActualValues[1]
//     Term 21 (AT2050-0500)/CC Inputs/Current actual value Ch.3 <-> Data Pointer/CurrentActualValues[2]
//     Term 21 (AT2050-0500)/CC Inputs/Current actual value Ch.4 <-> Data Pointer/CurrentActualValues[3]
//     Term 21 (AT2050-0500)/CC Inputs/Current actual value Ch.5 <-> Data Pointer/CurrentActualValues[4]
//     Term 21 (AT2050-0500)/CC Inputs/Current actual value Ch.6 <-> Data Pointer/CurrentActualValues[5]
//     Term 21 (AT2050-0500)/CC Inputs/Current actual value Ch.7 <-> Data Pointer/CurrentActualValues[6]
//     Term 21 (AT2050-0500)/CC Inputs/Current actual value Ch.8 <-> Data Pointer/CurrentActualValues[7]
//     Term 21 (AT2050-0500)/CC Inputs/Current actual value Ch.9 <-> Data Pointer/CurrentActualValues[8]
//     Term 21 (AT2050-0500)/CC Inputs/Status <-> Data Pointer/Status
//     Term 21 (AT2050-0500)/CC Outputs/Control <-> Data Pointer/Control
//     Term 21 (AT2050-0500)/CC Outputs/Current setpoint value Ch.1 <-> Data Pointer/CurrentSetpointValues[0]
//     Term 21 (AT2050-0500)/CC Outputs/Current setpoint value Ch.10 <-> Data Pointer/CurrentSetpointValues[9]
//     Term 21 (AT2050-0500)/CC Outputs/Current setpoint value Ch.11 <-> Data Pointer/CurrentSetpointValues[10]
//     Term 21 (AT2050-0500)/CC Outputs/Current setpoint value Ch.12 <-> Data Pointer/CurrentSetpointValues[11]
//     Term 21 (AT2050-0500)/CC Outputs/Current setpoint value Ch.13 <-> Data Pointer/CurrentSetpointValues[12]
//     Term 21 (AT2050-0500)/CC Outputs/Current setpoint value Ch.14 <-> Data Pointer/CurrentSetpointValues[13]
//     Term 21 (AT2050-0500)/CC Outputs/Current setpoint value Ch.15 <-> Data Pointer/CurrentSetpointValues[14]
//     Term 21 (AT2050-0500)/CC Outputs/Current setpoint value Ch.2 <-> Data Pointer/CurrentSetpointValues[1]
//     Term 21 (AT2050-0500)/CC Outputs/Current setpoint value Ch.3 <-> Data Pointer/CurrentSetpointValues[2]
//     Term 21 (AT2050-0500)/CC Outputs/Current setpoint value Ch.4 <-> Data Pointer/CurrentSetpointValues[3]
//     Term 21 (AT2050-0500)/CC Outputs/Current setpoint value Ch.5 <-> Data Pointer/CurrentSetpointValues[4]
//     Term 21 (AT2050-0500)/CC Outputs/Current setpoint value Ch.6 <-> Data Pointer/CurrentSetpointValues[5]
//     Term 21 (AT2050-0500)/CC Outputs/Current setpoint value Ch.7 <-> Data Pointer/CurrentSetpointValues[6]
//     Term 21 (AT2050-0500)/CC Outputs/Current setpoint value Ch.8 <-> Data Pointer/CurrentSetpointValues[7]
//     Term 21 (AT2050-0500)/CC Outputs/Current setpoint value Ch.9 <-> Data Pointer/CurrentSetpointValues[8]
//     Term 21 (AT2050-0500)/Term 22 (AT2050-5500)/FB Inputs/Value Channel 01 <-> Data Pointer/RawPositionValues[0]
//     Term 21 (AT2050-0500)/Term 22 (AT2050-5500)/FB Inputs/Value Channel 02 <-> Data Pointer/RawPositionValues[1]
//     Term 21 (AT2050-0500)/Term 22 (AT2050-5500)/FB Inputs/Value Channel 03 <-> Data Pointer/RawPositionValues[2]
//     Term 21 (AT2050-0500)/Term 22 (AT2050-5500)/FB Inputs/Value Channel 04 <-> Data Pointer/RawPositionValues[3]
//     Term 21 (AT2050-0500)/Term 22 (AT2050-5500)/FB Inputs/Value Channel 05 <-> Data Pointer/RawPositionValues[4]
//     Term 21 (AT2050-0500)/Term 22 (AT2050-5500)/FB Inputs/Value Channel 06 <-> Data Pointer/RawPositionValues[5]
//     Term 21 (AT2050-0500)/Term 22 (AT2050-5500)/FB Inputs/Value Channel 07 <-> Data Pointer/RawPositionValues[6]
//     Term 21 (AT2050-0500)/Term 22 (AT2050-5500)/FB Inputs/Value Channel 08 <-> Data Pointer/RawPositionValues[7]
//     Term 21 (AT2050-0500)/Term 22 (AT2050-5500)/FB Inputs/Value Channel 09 <-> Data Pointer/RawPositionValues[8]
//     Term 21 (AT2050-0500)/Term 22 (AT2050-5500)/FB Inputs/Value Channel 10 <-> Data Pointer/RawPositionValues[9]
//     Term 21 (AT2050-0500)/Term 22 (AT2050-5500)/FB Inputs/Value Channel 11 <-> Data Pointer/RawPositionValues[10]
//     Term 21 (AT2050-0500)/Term 22 (AT2050-5500)/FB Inputs/Value Channel 12 <-> Data Pointer/RawPositionValues[11]
//     Term 21 (AT2050-0500)/Term 22 (AT2050-5500)/FB Inputs/Value Channel 13 <-> Data Pointer/RawPositionValues[12]
//     Term 21 (AT2050-0500)/Term 22 (AT2050-5500)/FB Inputs/Value Channel 14 <-> Data Pointer/RawPositionValues[13]
//     Term 21 (AT2050-0500)/Term 22 (AT2050-5500)/FB Inputs/Value Channel 15 <-> Data Pointer/RawPositionValues[14]
//     Term 21 (AT2050-0500)/Term 22 (AT2050-5500)/FB Inputs/Value Channel 16 <-> Data Pointer/RawPositionValues[15]
//     Term 21 (AT2050-0500)/Term 22 (AT2050-5500)/FB Inputs/Value Channel 17 <-> Data Pointer/RawPositionValues[16]
//     Term 21 (AT2050-0500)/Term 22 (AT2050-5500)/FB Inputs/Value Channel 18 <-> Data Pointer/RawPositionValues[17]
//     Term 21 (AT2050-0500)/Term 22 (AT2050-5500)/FB Inputs/Value Channel 19 <-> Data Pointer/RawPositionValues[18]
//     Term 21 (AT2050-0500)/Term 22 (AT2050-5500)/FB Inputs/Value Channel 20 <-> Data Pointer/RawPositionValues[19]
//     Term 21 (AT2050-0500)/Term 22 (AT2050-5500)/FB Inputs/Value Channel 21 <-> Data Pointer/RawPositionValues[20]
//     Term 21 (AT2050-0500)/Term 22 (AT2050-5500)/FB Inputs/Value Channel 22 <-> Data Pointer/RawPositionValues[21]
//     Term 21 (AT2050-0500)/Term 22 (AT2050-5500)/FB Inputs/Value Channel 23 <-> Data Pointer/RawPositionValues[22]
//     Term 21 (AT2050-0500)/Term 22 (AT2050-5500)/FB Inputs/Value Channel 24 <-> Data Pointer/RawPositionValues[23]
//     Term 21 (AT2050-0500)/Term 22 (AT2050-5500)/FB Inputs/Value Channel 25 <-> Data Pointer/RawPositionValues[24]
//     Term 21 (AT2050-0500)/Term 22 (AT2050-5500)/FB Inputs/Value Channel 26 <-> Data Pointer/RawPositionValues[25]
//     Term 21 (AT2050-0500)/Term 22 (AT2050-5500)/FB Inputs/Value Channel 27 <-> Data Pointer/RawPositionValues[26]
//     Term 21 (AT2050-0500)/Term 22 (AT2050-5500)/FB Inputs/Value Channel 28 <-> Data Pointer/RawPositionValues[27]
//     Term 21 (AT2050-0500)/Term 22 (AT2050-5500)/FB Inputs/Value Channel 29 <-> Data Pointer/RawPositionValues[28]
//     Term 21 (AT2050-0500)/Term 22 (AT2050-5500)/FB Inputs/Value Channel 30 <-> Data Pointer/RawPositionValues[29]
//     Term 21 (AT2050-0500)/Term 22 (AT2050-5500)/FB Inputs/Value Channel 31 <-> Data Pointer/RawPositionValues[30]
//     Term 21 (AT2050-0500)/Term 22 (AT2050-5500)/FB Inputs/Value Channel 32 <-> Data Pointer/RawPositionValues[31]
//   Device 2 <-> TcCOM Objects/XtsProcessingUnit 1/Part 1/Module 12
//     Term 23 (AT2050-0501)/CC Inputs/Current actual value Ch.1 <-> Data Pointer/CurrentActualValues[0]
//     Term 23 (AT2050-0501)/CC Inputs/Current actual value Ch.10 <-> Data Pointer/CurrentActualValues[9]
//     Term 23 (AT2050-0501)/CC Inputs/Current actual value Ch.11 <-> Data Pointer/CurrentActualValues[10]
//     Term 23 (AT2050-0501)/CC Inputs/Current actual value Ch.12 <-> Data Pointer/CurrentActualValues[11]
//     Term 23 (AT2050-0501)/CC Inputs/Current actual value Ch.13 <-> Data Pointer/CurrentActualValues[12]
//     Term 23 (AT2050-0501)/CC Inputs/Current actual value Ch.14 <-> Data Pointer/CurrentActualValues[13]
//     Term 23 (AT2050-0501)/CC Inputs/Current actual value Ch.15 <-> Data Pointer/CurrentActualValues[14]
//     Term 23 (AT2050-0501)/CC Inputs/Current actual value Ch.2 <-> Data Pointer/CurrentActualValues[1]
//     Term 23 (AT2050-0501)/CC Inputs/Current actual value Ch.3 <-> Data Pointer/CurrentActualValues[2]
//     Term 23 (AT2050-0501)/CC Inputs/Current actual value Ch.4 <-> Data Pointer/CurrentActualValues[3]
//     Term 23 (AT2050-0501)/CC Inputs/Current actual value Ch.5 <-> Data Pointer/CurrentActualValues[4]
//     Term 23 (AT2050-0501)/CC Inputs/Current actual value Ch.6 <-> Data Pointer/CurrentActualValues[5]
//     Term 23 (AT2050-0501)/CC Inputs/Current actual value Ch.7 <-> Data Pointer/CurrentActualValues[6]
//     Term 23 (AT2050-0501)/CC Inputs/Current actual value Ch.8 <-> Data Pointer/CurrentActualValues[7]
//     Term 23 (AT2050-0501)/CC Inputs/Current actual value Ch.9 <-> Data Pointer/CurrentActualValues[8]
//     Term 23 (AT2050-0501)/CC Inputs/Status <-> Data Pointer/Status
//     Term 23 (AT2050-0501)/CC Outputs/Control <-> Data Pointer/Control
//     Term 23 (AT2050-0501)/CC Outputs/Current setpoint value Ch.1 <-> Data Pointer/CurrentSetpointValues[0]
//     Term 23 (AT2050-0501)/CC Outputs/Current setpoint value Ch.10 <-> Data Pointer/CurrentSetpointValues[9]
//     Term 23 (AT2050-0501)/CC Outputs/Current setpoint value Ch.11 <-> Data Pointer/CurrentSetpointValues[10]
//     Term 23 (AT2050-0501)/CC Outputs/Current setpoint value Ch.12 <-> Data Pointer/CurrentSetpointValues[11]
//     Term 23 (AT2050-0501)/CC Outputs/Current setpoint value Ch.13 <-> Data Pointer/CurrentSetpointValues[12]
//     Term 23 (AT2050-0501)/CC Outputs/Current setpoint value Ch.14 <-> Data Pointer/CurrentSetpointValues[13]
//     Term 23 (AT2050-0501)/CC Outputs/Current setpoint value Ch.15 <-> Data Pointer/CurrentSetpointValues[14]
//     Term 23 (AT2050-0501)/CC Outputs/Current setpoint value Ch.2 <-> Data Pointer/CurrentSetpointValues[1]
//     Term 23 (AT2050-0501)/CC Outputs/Current setpoint value Ch.3 <-> Data Pointer/CurrentSetpointValues[2]
//     Term 23 (AT2050-0501)/CC Outputs/Current setpoint value Ch.4 <-> Data Pointer/CurrentSetpointValues[3]
//     Term 23 (AT2050-0501)/CC Outputs/Current setpoint value Ch.5 <-> Data Pointer/CurrentSetpointValues[4]
//     Term 23 (AT2050-0501)/CC Outputs/Current setpoint value Ch.6 <-> Data Pointer/CurrentSetpointValues[5]
//     Term 23 (AT2050-0501)/CC Outputs/Current setpoint value Ch.7 <-> Data Pointer/CurrentSetpointValues[6]
//     Term 23 (AT2050-0501)/CC Outputs/Current setpoint value Ch.8 <-> Data Pointer/CurrentSetpointValues[7]
//     Term 23 (AT2050-0501)/CC Outputs/Current setpoint value Ch.9 <-> Data Pointer/CurrentSetpointValues[8]
//     Term 23 (AT2050-0501)/Term 24 (AT2050-5501)/FB Inputs/Value Channel 01 <-> Data Pointer/RawPositionValues[0]
//     Term 23 (AT2050-0501)/Term 24 (AT2050-5501)/FB Inputs/Value Channel 02 <-> Data Pointer/RawPositionValues[1]
//     Term 23 (AT2050-0501)/Term 24 (AT2050-5501)/FB Inputs/Value Channel 03 <-> Data Pointer/RawPositionValues[2]
//     Term 23 (AT2050-0501)/Term 24 (AT2050-5501)/FB Inputs/Value Channel 04 <-> Data Pointer/RawPositionValues[3]
//     Term 23 (AT2050-0501)/Term 24 (AT2050-5501)/FB Inputs/Value Channel 05 <-> Data Pointer/RawPositionValues[4]
//     Term 23 (AT2050-0501)/Term 24 (AT2050-5501)/FB Inputs/Value Channel 06 <-> Data Pointer/RawPositionValues[5]
//     Term 23 (AT2050-0501)/Term 24 (AT2050-5501)/FB Inputs/Value Channel 07 <-> Data Pointer/RawPositionValues[6]
//     Term 23 (AT2050-0501)/Term 24 (AT2050-5501)/FB Inputs/Value Channel 08 <-> Data Pointer/RawPositionValues[7]
//     Term 23 (AT2050-0501)/Term 24 (AT2050-5501)/FB Inputs/Value Channel 09 <-> Data Pointer/RawPositionValues[8]
//     Term 23 (AT2050-0501)/Term 24 (AT2050-5501)/FB Inputs/Value Channel 10 <-> Data Pointer/RawPositionValues[9]
//     Term 23 (AT2050-0501)/Term 24 (AT2050-5501)/FB Inputs/Value Channel 11 <-> Data Pointer/RawPositionValues[10]
//     Term 23 (AT2050-0501)/Term 24 (AT2050-5501)/FB Inputs/Value Channel 12 <-> Data Pointer/RawPositionValues[11]
//     Term 23 (AT2050-0501)/Term 24 (AT2050-5501)/FB Inputs/Value Channel 13 <-> Data Pointer/RawPositionValues[12]
//     Term 23 (AT2050-0501)/Term 24 (AT2050-5501)/FB Inputs/Value Channel 14 <-> Data Pointer/RawPositionValues[13]
//     Term 23 (AT2050-0501)/Term 24 (AT2050-5501)/FB Inputs/Value Channel 15 <-> Data Pointer/RawPositionValues[14]
//     Term 23 (AT2050-0501)/Term 24 (AT2050-5501)/FB Inputs/Value Channel 16 <-> Data Pointer/RawPositionValues[15]
//     Term 23 (AT2050-0501)/Term 24 (AT2050-5501)/FB Inputs/Value Channel 17 <-> Data Pointer/RawPositionValues[16]
//     Term 23 (AT2050-0501)/Term 24 (AT2050-5501)/FB Inputs/Value Channel 18 <-> Data Pointer/RawPositionValues[17]
//     Term 23 (AT2050-0501)/Term 24 (AT2050-5501)/FB Inputs/Value Channel 19 <-> Data Pointer/RawPositionValues[18]
//     Term 23 (AT2050-0501)/Term 24 (AT2050-5501)/FB Inputs/Value Channel 20 <-> Data Pointer/RawPositionValues[19]
//     Term 23 (AT2050-0501)/Term 24 (AT2050-5501)/FB Inputs/Value Channel 21 <-> Data Pointer/RawPositionValues[20]
//     Term 23 (AT2050-0501)/Term 24 (AT2050-5501)/FB Inputs/Value Channel 22 <-> Data Pointer/RawPositionValues[21]
//     Term 23 (AT2050-0501)/Term 24 (AT2050-5501)/FB Inputs/Value Channel 23 <-> Data Pointer/RawPositionValues[22]
//     Term 23 (AT2050-0501)/Term 24 (AT2050-5501)/FB Inputs/Value Channel 24 <-> Data Pointer/RawPositionValues[23]
//     Term 23 (AT2050-0501)/Term 24 (AT2050-5501)/FB Inputs/Value Channel 25 <-> Data Pointer/RawPositionValues[24]
//     Term 23 (AT2050-0501)/Term 24 (AT2050-5501)/FB Inputs/Value Channel 26 <-> Data Pointer/RawPositionValues[25]
//     Term 23 (AT2050-0501)/Term 24 (AT2050-5501)/FB Inputs/Value Channel 27 <-> Data Pointer/RawPositionValues[26]
//     Term 23 (AT2050-0501)/Term 24 (AT2050-5501)/FB Inputs/Value Channel 28 <-> Data Pointer/RawPositionValues[27]
//     Term 23 (AT2050-0501)/Term 24 (AT2050-5501)/FB Inputs/Value Channel 29 <-> Data Pointer/RawPositionValues[28]
//     Term 23 (AT2050-0501)/Term 24 (AT2050-5501)/FB Inputs/Value Channel 30 <-> Data Pointer/RawPositionValues[29]
//     Term 23 (AT2050-0501)/Term 24 (AT2050-5501)/FB Inputs/Value Channel 31 <-> Data Pointer/RawPositionValues[30]
//     Term 23 (AT2050-0501)/Term 24 (AT2050-5501)/FB Inputs/Value Channel 32 <-> Data Pointer/RawPositionValues[31]
//   Device 2 <-> TcCOM Objects/XtsProcessingUnit 1/Part 1/Module 7
//     Term 13 (AT2001-0250)/CC Inputs/Current actual value Ch.1 <-> Data Pointer/CurrentActualValues[0]
//     Term 13 (AT2001-0250)/CC Inputs/Current actual value Ch.10 <-> Data Pointer/CurrentActualValues[9]
//     Term 13 (AT2001-0250)/CC Inputs/Current actual value Ch.11 <-> Data Pointer/CurrentActualValues[10]
//     Term 13 (AT2001-0250)/CC Inputs/Current actual value Ch.12 <-> Data Pointer/CurrentActualValues[11]
//     Term 13 (AT2001-0250)/CC Inputs/Current actual value Ch.13 <-> Data Pointer/CurrentActualValues[12]
//     Term 13 (AT2001-0250)/CC Inputs/Current actual value Ch.14 <-> Data Pointer/CurrentActualValues[13]
//     Term 13 (AT2001-0250)/CC Inputs/Current actual value Ch.15 <-> Data Pointer/CurrentActualValues[14]
//     Term 13 (AT2001-0250)/CC Inputs/Current actual value Ch.2 <-> Data Pointer/CurrentActualValues[1]
//     Term 13 (AT2001-0250)/CC Inputs/Current actual value Ch.3 <-> Data Pointer/CurrentActualValues[2]
//     Term 13 (AT2001-0250)/CC Inputs/Current actual value Ch.4 <-> Data Pointer/CurrentActualValues[3]
//     Term 13 (AT2001-0250)/CC Inputs/Current actual value Ch.5 <-> Data Pointer/CurrentActualValues[4]
//     Term 13 (AT2001-0250)/CC Inputs/Current actual value Ch.6 <-> Data Pointer/CurrentActualValues[5]
//     Term 13 (AT2001-0250)/CC Inputs/Current actual value Ch.7 <-> Data Pointer/CurrentActualValues[6]
//     Term 13 (AT2001-0250)/CC Inputs/Current actual value Ch.8 <-> Data Pointer/CurrentActualValues[7]
//     Term 13 (AT2001-0250)/CC Inputs/Current actual value Ch.9 <-> Data Pointer/CurrentActualValues[8]
//     Term 13 (AT2001-0250)/CC Inputs/Status <-> Data Pointer/Status
//     Term 13 (AT2001-0250)/CC Outputs/Control <-> Data Pointer/Control
//     Term 13 (AT2001-0250)/CC Outputs/Current setpoint value Ch.1 <-> Data Pointer/CurrentSetpointValues[0]
//     Term 13 (AT2001-0250)/CC Outputs/Current setpoint value Ch.10 <-> Data Pointer/CurrentSetpointValues[9]
//     Term 13 (AT2001-0250)/CC Outputs/Current setpoint value Ch.11 <-> Data Pointer/CurrentSetpointValues[10]
//     Term 13 (AT2001-0250)/CC Outputs/Current setpoint value Ch.12 <-> Data Pointer/CurrentSetpointValues[11]
//     Term 13 (AT2001-0250)/CC Outputs/Current setpoint value Ch.13 <-> Data Pointer/CurrentSetpointValues[12]
//     Term 13 (AT2001-0250)/CC Outputs/Current setpoint value Ch.14 <-> Data Pointer/CurrentSetpointValues[13]
//     Term 13 (AT2001-0250)/CC Outputs/Current setpoint value Ch.15 <-> Data Pointer/CurrentSetpointValues[14]
//     Term 13 (AT2001-0250)/CC Outputs/Current setpoint value Ch.2 <-> Data Pointer/CurrentSetpointValues[1]
//     Term 13 (AT2001-0250)/CC Outputs/Current setpoint value Ch.3 <-> Data Pointer/CurrentSetpointValues[2]
//     Term 13 (AT2001-0250)/CC Outputs/Current setpoint value Ch.4 <-> Data Pointer/CurrentSetpointValues[3]
//     Term 13 (AT2001-0250)/CC Outputs/Current setpoint value Ch.5 <-> Data Pointer/CurrentSetpointValues[4]
//     Term 13 (AT2001-0250)/CC Outputs/Current setpoint value Ch.6 <-> Data Pointer/CurrentSetpointValues[5]
//     Term 13 (AT2001-0250)/CC Outputs/Current setpoint value Ch.7 <-> Data Pointer/CurrentSetpointValues[6]
//     Term 13 (AT2001-0250)/CC Outputs/Current setpoint value Ch.8 <-> Data Pointer/CurrentSetpointValues[7]
//     Term 13 (AT2001-0250)/CC Outputs/Current setpoint value Ch.9 <-> Data Pointer/CurrentSetpointValues[8]
//     Term 13 (AT2001-0250)/Term 14 (AT2001-5250)/FB Inputs/Value Channel 01 <-> Data Pointer/RawPositionValues[0]
//     Term 13 (AT2001-0250)/Term 14 (AT2001-5250)/FB Inputs/Value Channel 02 <-> Data Pointer/RawPositionValues[1]
//     Term 13 (AT2001-0250)/Term 14 (AT2001-5250)/FB Inputs/Value Channel 03 <-> Data Pointer/RawPositionValues[2]
//     Term 13 (AT2001-0250)/Term 14 (AT2001-5250)/FB Inputs/Value Channel 04 <-> Data Pointer/RawPositionValues[3]
//     Term 13 (AT2001-0250)/Term 14 (AT2001-5250)/FB Inputs/Value Channel 05 <-> Data Pointer/RawPositionValues[4]
//     Term 13 (AT2001-0250)/Term 14 (AT2001-5250)/FB Inputs/Value Channel 06 <-> Data Pointer/RawPositionValues[5]
//     Term 13 (AT2001-0250)/Term 14 (AT2001-5250)/FB Inputs/Value Channel 07 <-> Data Pointer/RawPositionValues[6]
//     Term 13 (AT2001-0250)/Term 14 (AT2001-5250)/FB Inputs/Value Channel 08 <-> Data Pointer/RawPositionValues[7]
//     Term 13 (AT2001-0250)/Term 14 (AT2001-5250)/FB Inputs/Value Channel 09 <-> Data Pointer/RawPositionValues[8]
//     Term 13 (AT2001-0250)/Term 14 (AT2001-5250)/FB Inputs/Value Channel 10 <-> Data Pointer/RawPositionValues[9]
//     Term 13 (AT2001-0250)/Term 14 (AT2001-5250)/FB Inputs/Value Channel 11 <-> Data Pointer/RawPositionValues[10]
//     Term 13 (AT2001-0250)/Term 14 (AT2001-5250)/FB Inputs/Value Channel 12 <-> Data Pointer/RawPositionValues[11]
//     Term 13 (AT2001-0250)/Term 14 (AT2001-5250)/FB Inputs/Value Channel 13 <-> Data Pointer/RawPositionValues[12]
//     Term 13 (AT2001-0250)/Term 14 (AT2001-5250)/FB Inputs/Value Channel 14 <-> Data Pointer/RawPositionValues[13]
//     Term 13 (AT2001-0250)/Term 14 (AT2001-5250)/FB Inputs/Value Channel 15 <-> Data Pointer/RawPositionValues[14]
//     Term 13 (AT2001-0250)/Term 14 (AT2001-5250)/FB Inputs/Value Channel 16 <-> Data Pointer/RawPositionValues[15]
//     Term 13 (AT2001-0250)/Term 14 (AT2001-5250)/FB Inputs/Value Channel 17 <-> Data Pointer/RawPositionValues[16]
//     Term 13 (AT2001-0250)/Term 14 (AT2001-5250)/FB Inputs/Value Channel 18 <-> Data Pointer/RawPositionValues[17]
//     Term 13 (AT2001-0250)/Term 14 (AT2001-5250)/FB Inputs/Value Channel 19 <-> Data Pointer/RawPositionValues[18]
//     Term 13 (AT2001-0250)/Term 14 (AT2001-5250)/FB Inputs/Value Channel 20 <-> Data Pointer/RawPositionValues[19]
//     Term 13 (AT2001-0250)/Term 14 (AT2001-5250)/FB Inputs/Value Channel 21 <-> Data Pointer/RawPositionValues[20]
//     Term 13 (AT2001-0250)/Term 14 (AT2001-5250)/FB Inputs/Value Channel 22 <-> Data Pointer/RawPositionValues[21]
//     Term 13 (AT2001-0250)/Term 14 (AT2001-5250)/FB Inputs/Value Channel 23 <-> Data Pointer/RawPositionValues[22]
//     Term 13 (AT2001-0250)/Term 14 (AT2001-5250)/FB Inputs/Value Channel 24 <-> Data Pointer/RawPositionValues[23]
//     Term 13 (AT2001-0250)/Term 14 (AT2001-5250)/FB Inputs/Value Channel 25 <-> Data Pointer/RawPositionValues[24]
//     Term 13 (AT2001-0250)/Term 14 (AT2001-5250)/FB Inputs/Value Channel 26 <-> Data Pointer/RawPositionValues[25]
//     Term 13 (AT2001-0250)/Term 14 (AT2001-5250)/FB Inputs/Value Channel 27 <-> Data Pointer/RawPositionValues[26]
//     Term 13 (AT2001-0250)/Term 14 (AT2001-5250)/FB Inputs/Value Channel 28 <-> Data Pointer/RawPositionValues[27]
//     Term 13 (AT2001-0250)/Term 14 (AT2001-5250)/FB Inputs/Value Channel 29 <-> Data Pointer/RawPositionValues[28]
//     Term 13 (AT2001-0250)/Term 14 (AT2001-5250)/FB Inputs/Value Channel 30 <-> Data Pointer/RawPositionValues[29]
//     Term 13 (AT2001-0250)/Term 14 (AT2001-5250)/FB Inputs/Value Channel 31 <-> Data Pointer/RawPositionValues[30]
//     Term 13 (AT2001-0250)/Term 14 (AT2001-5250)/FB Inputs/Value Channel 32 <-> Data Pointer/RawPositionValues[31]
//   Device 2 <-> TcCOM Objects/XtsProcessingUnit 1/Part 1/Module 8
//     Term 15 (AT2000-0250)/CC Inputs/Current actual value Ch.1 <-> Data Pointer/CurrentActualValues[0]
//     Term 15 (AT2000-0250)/CC Inputs/Current actual value Ch.10 <-> Data Pointer/CurrentActualValues[9]
//     Term 15 (AT2000-0250)/CC Inputs/Current actual value Ch.11 <-> Data Pointer/CurrentActualValues[10]
//     Term 15 (AT2000-0250)/CC Inputs/Current actual value Ch.12 <-> Data Pointer/CurrentActualValues[11]
//     Term 15 (AT2000-0250)/CC Inputs/Current actual value Ch.13 <-> Data Pointer/CurrentActualValues[12]
//     Term 15 (AT2000-0250)/CC Inputs/Current actual value Ch.14 <-> Data Pointer/CurrentActualValues[13]
//     Term 15 (AT2000-0250)/CC Inputs/Current actual value Ch.15 <-> Data Pointer/CurrentActualValues[14]
//     Term 15 (AT2000-0250)/CC Inputs/Current actual value Ch.2 <-> Data Pointer/CurrentActualValues[1]
//     Term 15 (AT2000-0250)/CC Inputs/Current actual value Ch.3 <-> Data Pointer/CurrentActualValues[2]
//     Term 15 (AT2000-0250)/CC Inputs/Current actual value Ch.4 <-> Data Pointer/CurrentActualValues[3]
//     Term 15 (AT2000-0250)/CC Inputs/Current actual value Ch.5 <-> Data Pointer/CurrentActualValues[4]
//     Term 15 (AT2000-0250)/CC Inputs/Current actual value Ch.6 <-> Data Pointer/CurrentActualValues[5]
//     Term 15 (AT2000-0250)/CC Inputs/Current actual value Ch.7 <-> Data Pointer/CurrentActualValues[6]
//     Term 15 (AT2000-0250)/CC Inputs/Current actual value Ch.8 <-> Data Pointer/CurrentActualValues[7]
//     Term 15 (AT2000-0250)/CC Inputs/Current actual value Ch.9 <-> Data Pointer/CurrentActualValues[8]
//     Term 15 (AT2000-0250)/CC Inputs/Status <-> Data Pointer/Status
//     Term 15 (AT2000-0250)/CC Outputs/Control <-> Data Pointer/Control
//     Term 15 (AT2000-0250)/CC Outputs/Current setpoint value Ch.1 <-> Data Pointer/CurrentSetpointValues[0]
//     Term 15 (AT2000-0250)/CC Outputs/Current setpoint value Ch.10 <-> Data Pointer/CurrentSetpointValues[9]
//     Term 15 (AT2000-0250)/CC Outputs/Current setpoint value Ch.11 <-> Data Pointer/CurrentSetpointValues[10]
//     Term 15 (AT2000-0250)/CC Outputs/Current setpoint value Ch.12 <-> Data Pointer/CurrentSetpointValues[11]
//     Term 15 (AT2000-0250)/CC Outputs/Current setpoint value Ch.13 <-> Data Pointer/CurrentSetpointValues[12]
//     Term 15 (AT2000-0250)/CC Outputs/Current setpoint value Ch.14 <-> Data Pointer/CurrentSetpointValues[13]
//     Term 15 (AT2000-0250)/CC Outputs/Current setpoint value Ch.15 <-> Data Pointer/CurrentSetpointValues[14]
//     Term 15 (AT2000-0250)/CC Outputs/Current setpoint value Ch.2 <-> Data Pointer/CurrentSetpointValues[1]
//     Term 15 (AT2000-0250)/CC Outputs/Current setpoint value Ch.3 <-> Data Pointer/CurrentSetpointValues[2]
//     Term 15 (AT2000-0250)/CC Outputs/Current setpoint value Ch.4 <-> Data Pointer/CurrentSetpointValues[3]
//     Term 15 (AT2000-0250)/CC Outputs/Current setpoint value Ch.5 <-> Data Pointer/CurrentSetpointValues[4]
//     Term 15 (AT2000-0250)/CC Outputs/Current setpoint value Ch.6 <-> Data Pointer/CurrentSetpointValues[5]
//     Term 15 (AT2000-0250)/CC Outputs/Current setpoint value Ch.7 <-> Data Pointer/CurrentSetpointValues[6]
//     Term 15 (AT2000-0250)/CC Outputs/Current setpoint value Ch.8 <-> Data Pointer/CurrentSetpointValues[7]
//     Term 15 (AT2000-0250)/CC Outputs/Current setpoint value Ch.9 <-> Data Pointer/CurrentSetpointValues[8]
//     Term 15 (AT2000-0250)/Term 16 (AT2000-5250)/FB Inputs/Value Channel 01 <-> Data Pointer/RawPositionValues[0]
//     Term 15 (AT2000-0250)/Term 16 (AT2000-5250)/FB Inputs/Value Channel 02 <-> Data Pointer/RawPositionValues[1]
//     Term 15 (AT2000-0250)/Term 16 (AT2000-5250)/FB Inputs/Value Channel 03 <-> Data Pointer/RawPositionValues[2]
//     Term 15 (AT2000-0250)/Term 16 (AT2000-5250)/FB Inputs/Value Channel 04 <-> Data Pointer/RawPositionValues[3]
//     Term 15 (AT2000-0250)/Term 16 (AT2000-5250)/FB Inputs/Value Channel 05 <-> Data Pointer/RawPositionValues[4]
//     Term 15 (AT2000-0250)/Term 16 (AT2000-5250)/FB Inputs/Value Channel 06 <-> Data Pointer/RawPositionValues[5]
//     Term 15 (AT2000-0250)/Term 16 (AT2000-5250)/FB Inputs/Value Channel 07 <-> Data Pointer/RawPositionValues[6]
//     Term 15 (AT2000-0250)/Term 16 (AT2000-5250)/FB Inputs/Value Channel 08 <-> Data Pointer/RawPositionValues[7]
//     Term 15 (AT2000-0250)/Term 16 (AT2000-5250)/FB Inputs/Value Channel 09 <-> Data Pointer/RawPositionValues[8]
//     Term 15 (AT2000-0250)/Term 16 (AT2000-5250)/FB Inputs/Value Channel 10 <-> Data Pointer/RawPositionValues[9]
//     Term 15 (AT2000-0250)/Term 16 (AT2000-5250)/FB Inputs/Value Channel 11 <-> Data Pointer/RawPositionValues[10]
//     Term 15 (AT2000-0250)/Term 16 (AT2000-5250)/FB Inputs/Value Channel 12 <-> Data Pointer/RawPositionValues[11]
//     Term 15 (AT2000-0250)/Term 16 (AT2000-5250)/FB Inputs/Value Channel 13 <-> Data Pointer/RawPositionValues[12]
//     Term 15 (AT2000-0250)/Term 16 (AT2000-5250)/FB Inputs/Value Channel 14 <-> Data Pointer/RawPositionValues[13]
//     Term 15 (AT2000-0250)/Term 16 (AT2000-5250)/FB Inputs/Value Channel 15 <-> Data Pointer/RawPositionValues[14]
//     Term 15 (AT2000-0250)/Term 16 (AT2000-5250)/FB Inputs/Value Channel 16 <-> Data Pointer/RawPositionValues[15]
//     Term 15 (AT2000-0250)/Term 16 (AT2000-5250)/FB Inputs/Value Channel 17 <-> Data Pointer/RawPositionValues[16]
//     Term 15 (AT2000-0250)/Term 16 (AT2000-5250)/FB Inputs/Value Channel 18 <-> Data Pointer/RawPositionValues[17]
//     Term 15 (AT2000-0250)/Term 16 (AT2000-5250)/FB Inputs/Value Channel 19 <-> Data Pointer/RawPositionValues[18]
//     Term 15 (AT2000-0250)/Term 16 (AT2000-5250)/FB Inputs/Value Channel 20 <-> Data Pointer/RawPositionValues[19]
//     Term 15 (AT2000-0250)/Term 16 (AT2000-5250)/FB Inputs/Value Channel 21 <-> Data Pointer/RawPositionValues[20]
//     Term 15 (AT2000-0250)/Term 16 (AT2000-5250)/FB Inputs/Value Channel 22 <-> Data Pointer/RawPositionValues[21]
//     Term 15 (AT2000-0250)/Term 16 (AT2000-5250)/FB Inputs/Value Channel 23 <-> Data Pointer/RawPositionValues[22]
//     Term 15 (AT2000-0250)/Term 16 (AT2000-5250)/FB Inputs/Value Channel 24 <-> Data Pointer/RawPositionValues[23]
//     Term 15 (AT2000-0250)/Term 16 (AT2000-5250)/FB Inputs/Value Channel 25 <-> Data Pointer/RawPositionValues[24]
//     Term 15 (AT2000-0250)/Term 16 (AT2000-5250)/FB Inputs/Value Channel 26 <-> Data Pointer/RawPositionValues[25]
//     Term 15 (AT2000-0250)/Term 16 (AT2000-5250)/FB Inputs/Value Channel 27 <-> Data Pointer/RawPositionValues[26]
//     Term 15 (AT2000-0250)/Term 16 (AT2000-5250)/FB Inputs/Value Channel 28 <-> Data Pointer/RawPositionValues[27]
//     Term 15 (AT2000-0250)/Term 16 (AT2000-5250)/FB Inputs/Value Channel 29 <-> Data Pointer/RawPositionValues[28]
//     Term 15 (AT2000-0250)/Term 16 (AT2000-5250)/FB Inputs/Value Channel 30 <-> Data Pointer/RawPositionValues[29]
//     Term 15 (AT2000-0250)/Term 16 (AT2000-5250)/FB Inputs/Value Channel 31 <-> Data Pointer/RawPositionValues[30]
//     Term 15 (AT2000-0250)/Term 16 (AT2000-5250)/FB Inputs/Value Channel 32 <-> Data Pointer/RawPositionValues[31]
//   Device 2 <-> TcCOM Objects/XtsProcessingUnit 1/Part 1/Module 9
//     Term 17 (AT2000-0250)/CC Inputs/Current actual value Ch.1 <-> Data Pointer/CurrentActualValues[0]
//     Term 17 (AT2000-0250)/CC Inputs/Current actual value Ch.10 <-> Data Pointer/CurrentActualValues[9]
//     Term 17 (AT2000-0250)/CC Inputs/Current actual value Ch.11 <-> Data Pointer/CurrentActualValues[10]
//     Term 17 (AT2000-0250)/CC Inputs/Current actual value Ch.12 <-> Data Pointer/CurrentActualValues[11]
//     Term 17 (AT2000-0250)/CC Inputs/Current actual value Ch.13 <-> Data Pointer/CurrentActualValues[12]
//     Term 17 (AT2000-0250)/CC Inputs/Current actual value Ch.14 <-> Data Pointer/CurrentActualValues[13]
//     Term 17 (AT2000-0250)/CC Inputs/Current actual value Ch.15 <-> Data Pointer/CurrentActualValues[14]
//     Term 17 (AT2000-0250)/CC Inputs/Current actual value Ch.2 <-> Data Pointer/CurrentActualValues[1]
//     Term 17 (AT2000-0250)/CC Inputs/Current actual value Ch.3 <-> Data Pointer/CurrentActualValues[2]
//     Term 17 (AT2000-0250)/CC Inputs/Current actual value Ch.4 <-> Data Pointer/CurrentActualValues[3]
//     Term 17 (AT2000-0250)/CC Inputs/Current actual value Ch.5 <-> Data Pointer/CurrentActualValues[4]
//     Term 17 (AT2000-0250)/CC Inputs/Current actual value Ch.6 <-> Data Pointer/CurrentActualValues[5]
//     Term 17 (AT2000-0250)/CC Inputs/Current actual value Ch.7 <-> Data Pointer/CurrentActualValues[6]
//     Term 17 (AT2000-0250)/CC Inputs/Current actual value Ch.8 <-> Data Pointer/CurrentActualValues[7]
//     Term 17 (AT2000-0250)/CC Inputs/Current actual value Ch.9 <-> Data Pointer/CurrentActualValues[8]
//     Term 17 (AT2000-0250)/CC Inputs/Status <-> Data Pointer/Status
//     Term 17 (AT2000-0250)/CC Outputs/Control <-> Data Pointer/Control
//     Term 17 (AT2000-0250)/CC Outputs/Current setpoint value Ch.1 <-> Data Pointer/CurrentSetpointValues[0]
//     Term 17 (AT2000-0250)/CC Outputs/Current setpoint value Ch.10 <-> Data Pointer/CurrentSetpointValues[9]
//     Term 17 (AT2000-0250)/CC Outputs/Current setpoint value Ch.11 <-> Data Pointer/CurrentSetpointValues[10]
//     Term 17 (AT2000-0250)/CC Outputs/Current setpoint value Ch.12 <-> Data Pointer/CurrentSetpointValues[11]
//     Term 17 (AT2000-0250)/CC Outputs/Current setpoint value Ch.13 <-> Data Pointer/CurrentSetpointValues[12]
//     Term 17 (AT2000-0250)/CC Outputs/Current setpoint value Ch.14 <-> Data Pointer/CurrentSetpointValues[13]
//     Term 17 (AT2000-0250)/CC Outputs/Current setpoint value Ch.15 <-> Data Pointer/CurrentSetpointValues[14]
//     Term 17 (AT2000-0250)/CC Outputs/Current setpoint value Ch.2 <-> Data Pointer/CurrentSetpointValues[1]
//     Term 17 (AT2000-0250)/CC Outputs/Current setpoint value Ch.3 <-> Data Pointer/CurrentSetpointValues[2]
//     Term 17 (AT2000-0250)/CC Outputs/Current setpoint value Ch.4 <-> Data Pointer/CurrentSetpointValues[3]
//     Term 17 (AT2000-0250)/CC Outputs/Current setpoint value Ch.5 <-> Data Pointer/CurrentSetpointValues[4]
//     Term 17 (AT2000-0250)/CC Outputs/Current setpoint value Ch.6 <-> Data Pointer/CurrentSetpointValues[5]
//     Term 17 (AT2000-0250)/CC Outputs/Current setpoint value Ch.7 <-> Data Pointer/CurrentSetpointValues[6]
//     Term 17 (AT2000-0250)/CC Outputs/Current setpoint value Ch.8 <-> Data Pointer/CurrentSetpointValues[7]
//     Term 17 (AT2000-0250)/CC Outputs/Current setpoint value Ch.9 <-> Data Pointer/CurrentSetpointValues[8]
//     Term 17 (AT2000-0250)/Term 18 (AT2000-5250)/FB Inputs/Value Channel 01 <-> Data Pointer/RawPositionValues[0]
//     Term 17 (AT2000-0250)/Term 18 (AT2000-5250)/FB Inputs/Value Channel 02 <-> Data Pointer/RawPositionValues[1]
//     Term 17 (AT2000-0250)/Term 18 (AT2000-5250)/FB Inputs/Value Channel 03 <-> Data Pointer/RawPositionValues[2]
//     Term 17 (AT2000-0250)/Term 18 (AT2000-5250)/FB Inputs/Value Channel 04 <-> Data Pointer/RawPositionValues[3]
//     Term 17 (AT2000-0250)/Term 18 (AT2000-5250)/FB Inputs/Value Channel 05 <-> Data Pointer/RawPositionValues[4]
//     Term 17 (AT2000-0250)/Term 18 (AT2000-5250)/FB Inputs/Value Channel 06 <-> Data Pointer/RawPositionValues[5]
//     Term 17 (AT2000-0250)/Term 18 (AT2000-5250)/FB Inputs/Value Channel 07 <-> Data Pointer/RawPositionValues[6]
//     Term 17 (AT2000-0250)/Term 18 (AT2000-5250)/FB Inputs/Value Channel 08 <-> Data Pointer/RawPositionValues[7]
//     Term 17 (AT2000-0250)/Term 18 (AT2000-5250)/FB Inputs/Value Channel 09 <-> Data Pointer/RawPositionValues[8]
//     Term 17 (AT2000-0250)/Term 18 (AT2000-5250)/FB Inputs/Value Channel 10 <-> Data Pointer/RawPositionValues[9]
//     Term 17 (AT2000-0250)/Term 18 (AT2000-5250)/FB Inputs/Value Channel 11 <-> Data Pointer/RawPositionValues[10]
//     Term 17 (AT2000-0250)/Term 18 (AT2000-5250)/FB Inputs/Value Channel 12 <-> Data Pointer/RawPositionValues[11]
//     Term 17 (AT2000-0250)/Term 18 (AT2000-5250)/FB Inputs/Value Channel 13 <-> Data Pointer/RawPositionValues[12]
//     Term 17 (AT2000-0250)/Term 18 (AT2000-5250)/FB Inputs/Value Channel 14 <-> Data Pointer/RawPositionValues[13]
//     Term 17 (AT2000-0250)/Term 18 (AT2000-5250)/FB Inputs/Value Channel 15 <-> Data Pointer/RawPositionValues[14]
//     Term 17 (AT2000-0250)/Term 18 (AT2000-5250)/FB Inputs/Value Channel 16 <-> Data Pointer/RawPositionValues[15]
//     Term 17 (AT2000-0250)/Term 18 (AT2000-5250)/FB Inputs/Value Channel 17 <-> Data Pointer/RawPositionValues[16]
//     Term 17 (AT2000-0250)/Term 18 (AT2000-5250)/FB Inputs/Value Channel 18 <-> Data Pointer/RawPositionValues[17]
//     Term 17 (AT2000-0250)/Term 18 (AT2000-5250)/FB Inputs/Value Channel 19 <-> Data Pointer/RawPositionValues[18]
//     Term 17 (AT2000-0250)/Term 18 (AT2000-5250)/FB Inputs/Value Channel 20 <-> Data Pointer/RawPositionValues[19]
//     Term 17 (AT2000-0250)/Term 18 (AT2000-5250)/FB Inputs/Value Channel 21 <-> Data Pointer/RawPositionValues[20]
//     Term 17 (AT2000-0250)/Term 18 (AT2000-5250)/FB Inputs/Value Channel 22 <-> Data Pointer/RawPositionValues[21]
//     Term 17 (AT2000-0250)/Term 18 (AT2000-5250)/FB Inputs/Value Channel 23 <-> Data Pointer/RawPositionValues[22]
//     Term 17 (AT2000-0250)/Term 18 (AT2000-5250)/FB Inputs/Value Channel 24 <-> Data Pointer/RawPositionValues[23]
//     Term 17 (AT2000-0250)/Term 18 (AT2000-5250)/FB Inputs/Value Channel 25 <-> Data Pointer/RawPositionValues[24]
//     Term 17 (AT2000-0250)/Term 18 (AT2000-5250)/FB Inputs/Value Channel 26 <-> Data Pointer/RawPositionValues[25]
//     Term 17 (AT2000-0250)/Term 18 (AT2000-5250)/FB Inputs/Value Channel 27 <-> Data Pointer/RawPositionValues[26]
//     Term 17 (AT2000-0250)/Term 18 (AT2000-5250)/FB Inputs/Value Channel 28 <-> Data Pointer/RawPositionValues[27]
//     Term 17 (AT2000-0250)/Term 18 (AT2000-5250)/FB Inputs/Value Channel 29 <-> Data Pointer/RawPositionValues[28]
//     Term 17 (AT2000-0250)/Term 18 (AT2000-5250)/FB Inputs/Value Channel 30 <-> Data Pointer/RawPositionValues[29]
//     Term 17 (AT2000-0250)/Term 18 (AT2000-5250)/FB Inputs/Value Channel 31 <-> Data Pointer/RawPositionValues[30]
//     Term 17 (AT2000-0250)/Term 18 (AT2000-5250)/FB Inputs/Value Channel 32 <-> Data Pointer/RawPositionValues[31]
//   NC-Task 1/Axes/Mover Axis 1 <-> TcCOM Objects/XtsProcessingUnit 1/Mover 1
//     SoftDrive 1/Data Pointer/InputPointer1 <-> Inputs/SoftDriveInput
//     SoftDrive 1/Data Pointer/OutputPointer1 <-> Outputs/SoftDriveOutput
//   NC-Task 1/Axes/Mover Axis 10 <-> TcCOM Objects/XtsProcessingUnit 1/Mover 10
//     SoftDrive 10/Data Pointer/InputPointer1 <-> Inputs/SoftDriveInput
//     SoftDrive 10/Data Pointer/OutputPointer1 <-> Outputs/SoftDriveOutput
//   NC-Task 1/Axes/Mover Axis 2 <-> TcCOM Objects/XtsProcessingUnit 1/Mover 2
//     SoftDrive 2/Data Pointer/InputPointer1 <-> Inputs/SoftDriveInput
//     SoftDrive 2/Data Pointer/OutputPointer1 <-> Outputs/SoftDriveOutput
//   NC-Task 1/Axes/Mover Axis 3 <-> TcCOM Objects/XtsProcessingUnit 1/Mover 3
//     SoftDrive 3/Data Pointer/InputPointer1 <-> Inputs/SoftDriveInput
//     SoftDrive 3/Data Pointer/OutputPointer1 <-> Outputs/SoftDriveOutput
//   NC-Task 1/Axes/Mover Axis 4 <-> TcCOM Objects/XtsProcessingUnit 1/Mover 4
//     SoftDrive 4/Data Pointer/InputPointer1 <-> Inputs/SoftDriveInput
//     SoftDrive 4/Data Pointer/OutputPointer1 <-> Outputs/SoftDriveOutput
//   NC-Task 1/Axes/Mover Axis 5 <-> TcCOM Objects/XtsProcessingUnit 1/Mover 5
//     SoftDrive 5/Data Pointer/InputPointer1 <-> Inputs/SoftDriveInput
//     SoftDrive 5/Data Pointer/OutputPointer1 <-> Outputs/SoftDriveOutput
//   NC-Task 1/Axes/Mover Axis 6 <-> TcCOM Objects/XtsProcessingUnit 1/Mover 6
//     SoftDrive 6/Data Pointer/InputPointer1 <-> Inputs/SoftDriveInput
//     SoftDrive 6/Data Pointer/OutputPointer1 <-> Outputs/SoftDriveOutput
//   NC-Task 1/Axes/Mover Axis 7 <-> TcCOM Objects/XtsProcessingUnit 1/Mover 7
//     SoftDrive 7/Data Pointer/InputPointer1 <-> Inputs/SoftDriveInput
//     SoftDrive 7/Data Pointer/OutputPointer1 <-> Outputs/SoftDriveOutput
//   NC-Task 1/Axes/Mover Axis 8 <-> TcCOM Objects/XtsProcessingUnit 1/Mover 8
//     SoftDrive 8/Data Pointer/InputPointer1 <-> Inputs/SoftDriveInput
//     SoftDrive 8/Data Pointer/OutputPointer1 <-> Outputs/SoftDriveOutput
//   NC-Task 1/Axes/Mover Axis 9 <-> TcCOM Objects/XtsProcessingUnit 1/Mover 9
//     SoftDrive 9/Data Pointer/InputPointer1 <-> Inputs/SoftDriveInput
//     SoftDrive 9/Data Pointer/OutputPointer1 <-> Outputs/SoftDriveOutput
//   PLC/PLC Instance <-> NC-Task 1/Axes/Mover Axis 1
//     PlcTask Inputs/MAIN.Machine.XPU.Movers[1]._Axis.NcToPlc <-> Outputs/ToPlc
//     PlcTask Outputs/MAIN.Machine.XPU.Movers[1]._Axis.PlcToNc <-> Inputs/FromPlc
//   PLC/PLC Instance <-> NC-Task 1/Axes/Mover Axis 10
//     PlcTask Inputs/MAIN.Machine.XPU.Movers[10]._Axis.NcToPlc <-> Outputs/ToPlc
//     PlcTask Outputs/MAIN.Machine.XPU.Movers[10]._Axis.PlcToNc <-> Inputs/FromPlc
//   PLC/PLC Instance <-> NC-Task 1/Axes/Mover Axis 2
//     PlcTask Inputs/MAIN.Machine.XPU.Movers[2]._Axis.NcToPlc <-> Outputs/ToPlc
//     PlcTask Outputs/MAIN.Machine.XPU.Movers[2]._Axis.PlcToNc <-> Inputs/FromPlc
//   PLC/PLC Instance <-> NC-Task 1/Axes/Mover Axis 3
//     PlcTask Inputs/MAIN.Machine.XPU.Movers[3]._Axis.NcToPlc <-> Outputs/ToPlc
//     PlcTask Outputs/MAIN.Machine.XPU.Movers[3]._Axis.PlcToNc <-> Inputs/FromPlc
//   PLC/PLC Instance <-> NC-Task 1/Axes/Mover Axis 4
//     PlcTask Inputs/MAIN.Machine.XPU.Movers[4]._Axis.NcToPlc <-> Outputs/ToPlc
//     PlcTask Outputs/MAIN.Machine.XPU.Movers[4]._Axis.PlcToNc <-> Inputs/FromPlc
//   PLC/PLC Instance <-> NC-Task 1/Axes/Mover Axis 5
//     PlcTask Inputs/MAIN.Machine.XPU.Movers[5]._Axis.NcToPlc <-> Outputs/ToPlc
//     PlcTask Outputs/MAIN.Machine.XPU.Movers[5]._Axis.PlcToNc <-> Inputs/FromPlc
//   PLC/PLC Instance <-> NC-Task 1/Axes/Mover Axis 6
